    CONST robtarget Target_5570:=[[241.834905648,46.985576036,25.649683148],[0.692516726,0.060687774,-0.040025667,0.717729422],[-2,0,-1,0],[9E+09,9E+09,9E+09,9E+09,9E+09,9E+09]];
    CONST robtarget Target_5580:=[[234.328319461,46.702749675,25.84956623],[0.692516726,0.060687774,-0.040025667,0.717729422],[-2,0,-1,0],[9E+09,9E+09,9E+09,9E+09,9E+09,9E+09]];
    CONST robtarget Target_5590:=[[234.035172753,46.711233475,25.857420102],[0.692516726,0.060687774,-0.040025666,0.717729422],[-2,0,-1,0],[9E+09,9E+09,9E+09,9E+09,9E+09,9E+09]];
    CONST robtarget Target_5600:=[[233.779548655,46.760188453,25.864370937],[0.692516726,0.060687774,-0.040025666,0.717729422],[-2,0,-1,0],[9E+09,9E+09,9E+09,9E+09,9E+09,9E+09]];
    CONST robtarget Target_5610:=[[233.561447167,46.849614606,25.870418733],[0.692516726,0.060687774,-0.040025666,0.717729422],[-1,-1,0,0],[9E+09,9E+09,9E+09,9E+09,9E+09,9E+09]];
    CONST robtarget Target_5620:=[[233.380868291,46.979511937,25.875563491],[0.692516726,0.060687774,-0.040025667,0.717729422],[-1,-1,0,0],[9E+09,9E+09,9E+09,9E+09,9E+09,9E+09]];
    CONST robtarget Target_5630:=[[233.237812023,47.149880444,25.879805211],[0.692516726,0.060687774,-0.040025666,0.717729422],[-1,-1,0,0],[9E+09,9E+09,9E+09,9E+09,9E+09,9E+09]];
    CONST robtarget Target_5640:=[[233.132278367,47.360720127,25.883143893],[0.692516726,0.060687774,-0.040025666,0.717729422],[-1,-1,0,0],[9E+09,9E+09,9E+09,9E+09,9E+09,9E+09]];
    CONST robtarget Target_5650:=[[233.064267321,47.612030988,25.885579537],[0.692516726,0.060687774,-0.040025667,0.717729422],[-1,-1,0,0],[9E+09,9E+09,9E+09,9E+09,9E+09,9E+09]];
    CONST robtarget Target_5660:=[[233.033778885,47.903813024,25.887112143],[0.692516726,0.060687774,-0.040025667,0.717729422],[-1,-1,0,0],[9E+09,9E+09,9E+09,9E+09,9E+09,9E+09]];
    CONST robtarget Target_5670:=[[232.563911843,60.405319209,25.930427697],[0.692516726,0.060687774,-0.040025667,0.717729422],[-1,-1,0,0],[9E+09,9E+09,9E+09,9E+09,9E+09,9E+09]];
    CONST robtarget Target_5680:=[[232.572411908,60.698570219,25.930922129],[0.692516726,0.060687774,-0.040025667,0.717729422],[-1,-1,0,0],[9E+09,9E+09,9E+09,9E+09,9E+09,9E+09]];
    CONST robtarget Target_5690:=[[232.621366367,60.954288,25.930243251],[0.692516726,0.060687774,-0.040025666,0.717729422],[-1,-1,0,0],[9E+09,9E+09,9E+09,9E+09,9E+09,9E+09]];
    CONST robtarget Target_5700:=[[232.710775218,61.172472552,25.928391064],[0.692516726,0.060687774,-0.040025667,0.717729422],[-1,-1,0,0],[9E+09,9E+09,9E+09,9E+09,9E+09,9E+09]];
    CONST robtarget Target_5710:=[[232.840638463,61.353123873,25.925365567],[0.692516726,0.060687774,-0.040025666,0.717729422],[-1,-1,0,0],[9E+09,9E+09,9E+09,9E+09,9E+09,9E+09]];
    CONST robtarget Target_5720:=[[233.0109561,61.496241965,25.92116676],[0.692516726,0.060687774,-0.040025667,0.717729422],[-1,-1,0,0],[9E+09,9E+09,9E+09,9E+09,9E+09,9E+09]];
    CONST robtarget Target_5730:=[[233.221728132,61.601826826,25.915794643],[0.692516726,0.060687774,-0.040025667,0.717729422],[-1,-1,0,0],[9E+09,9E+09,9E+09,9E+09,9E+09,9E+09]];
    CONST robtarget Target_5740:=[[233.472954556,61.669878459,25.909249216],[0.692516726,0.060687774,-0.040025666,0.717729422],[-1,-1,0,0],[9E+09,9E+09,9E+09,9E+09,9E+09,9E+09]];
    CONST robtarget Target_5750:=[[233.764635372,61.700396861,25.90153048],[0.692516726,0.060687774,-0.040025667,0.717729422],[-2,0,-1,0],[9E+09,9E+09,9E+09,9E+09,9E+09,9E+09]];
    CONST robtarget Target_5760:=[[237.507531532,61.841418315,25.801865785],[0.692516726,0.060687774,-0.040025667,0.717729422],[-2,0,-1,0],[9E+09,9E+09,9E+09,9E+09,9E+09,9E+09]];
    CONST robtarget Target_5770:=[[237.80067824,61.832934515,25.794011913],[0.692516726,0.060687774,-0.040025666,0.717729422],[-2,0,-1,0],[9E+09,9E+09,9E+09,9E+09,9E+09,9E+09]];
    CONST robtarget Target_5780:=[[238.056302338,61.783979538,25.787061079],[0.692516726,0.060687774,-0.040025666,0.717729422],[-2,0,-1,0],[9E+09,9E+09,9E+09,9E+09,9E+09,9E+09]];
    CONST robtarget Target_5790:=[[238.274403825,61.694553384,25.781013283],[0.692516726,0.060687774,-0.040025666,0.717729422],[-2,0,-1,0],[9E+09,9E+09,9E+09,9E+09,9E+09,9E+09]];
    CONST robtarget Target_5800:=[[238.454982703,61.564656054,25.775868524],[0.692516726,0.060687774,-0.040025667,0.717729422],[-2,0,-1,0],[9E+09,9E+09,9E+09,9E+09,9E+09,9E+09]];
    CONST robtarget Target_5810:=[[238.598038969,61.394287547,25.771626804],[0.692516726,0.060687774,-0.040025666,0.717729422],[-2,0,-1,0],[9E+09,9E+09,9E+09,9E+09,9E+09,9E+09]];
    CONST robtarget Target_5820:=[[238.703572626,61.183447863,25.768288122],[0.692516726,0.060687774,-0.040025666,0.717729422],[-2,0,-1,0],[9E+09,9E+09,9E+09,9E+09,9E+09,9E+09]];
    CONST robtarget Target_5830:=[[238.771583672,60.932137002,25.765852478],[0.692516726,0.060687774,-0.040025667,0.717729422],[-2,0,-1,0],[9E+09,9E+09,9E+09,9E+09,9E+09,9E+09]];
    CONST robtarget Target_5840:=[[238.802072109,60.640354966,25.764319872],[0.692516726,0.060687774,-0.040025667,0.717729422],[-2,0,-1,0],[9E+09,9E+09,9E+09,9E+09,9E+09,9E+09]];
    CONST robtarget Target_5850:=[[238.793572042,60.347103955,25.76382544],[0.692516726,0.060687774,-0.040025667,0.717729422],[-2,0,-1,0],[9E+09,9E+09,9E+09,9E+09,9E+09,9E+09]];
    CONST robtarget Target_5860:=[[238.744617584,60.091386175,25.764504318],[0.692516726,0.060687774,-0.040025666,0.717729422],[-2,0,-1,0],[9E+09,9E+09,9E+09,9E+09,9E+09,9E+09]];
    CONST robtarget Target_5870:=[[238.655208732,59.873201624,25.766356505],[0.692516726,0.060687774,-0.040025667,0.717729422],[-2,0,-1,0],[9E+09,9E+09,9E+09,9E+09,9E+09,9E+09]];
    CONST robtarget Target_5880:=[[238.525345488,59.692550302,25.769382002],[0.692516726,0.060687774,-0.040025666,0.717729422],[-2,0,-1,0],[9E+09,9E+09,9E+09,9E+09,9E+09,9E+09]];
    CONST robtarget Target_5890:=[[238.35502785,59.549432211,25.773580809],[0.692516726,0.060687774,-0.040025667,0.717729422],[-2,0,-1,0],[9E+09,9E+09,9E+09,9E+09,9E+09,9E+09]];
    CONST robtarget Target_5900:=[[238.14425582,59.443847349,25.778952926],[0.692516726,0.060687774,-0.040025667,0.717729422],[-2,0,-1,0],[9E+09,9E+09,9E+09,9E+09,9E+09,9E+09]];
    CONST robtarget Target_5910:=[[237.893029395,59.375795717,25.785498353],[0.692516726,0.060687774,-0.040025666,0.717729422],[-2,0,-1,0],[9E+09,9E+09,9E+09,9E+09,9E+09,9E+09]];
    CONST robtarget Target_5920:=[[237.601348578,59.345277314,25.793217089],[0.692516726,0.060687774,-0.040025667,0.717729422],[-2,0,-1,0],[9E+09,9E+09,9E+09,9E+09,9E+09,9E+09]];
    CONST robtarget Target_5930:=[[236.800025002,59.419067101,-4.195988229],[0.692516726,0.060687774,-0.040025667,0.717729422],[-2,0,-1,0],[9E+09,9E+09,9E+09,9E+09,9E+09,9E+09]];
    CONST robtarget Target_5940:=[[225.383702429,63.988284743,-3.879696752],[0.692516726,0.060687774,-0.040025667,0.717729422],[0,0,0,0],[9E+09,9E+09,9E+09,9E+09,9E+09,9E+09]];
    CONST robtarget Target_5950:=[[226.185026006,63.914494956,26.109508566],[0.692516726,0.060687774,-0.040025667,0.717729422],[0,0,0,0],[9E+09,9E+09,9E+09,9E+09,9E+09,9E+09]];
    CONST robtarget Target_5960:=[[226.478172714,63.906011155,26.101654694],[0.692516726,0.060687774,-0.040025666,0.717729422],[0,0,0,0],[9E+09,9E+09,9E+09,9E+09,9E+09,9E+09]];
    CONST robtarget Target_5970:=[[226.733796812,63.857056178,26.094703859],[0.692516726,0.060687774,-0.040025666,0.717729422],[0,0,0,0],[9E+09,9E+09,9E+09,9E+09,9E+09,9E+09]];
    CONST robtarget Target_5980:=[[226.951898299,63.767630024,26.088656063],[0.692516726,0.060687774,-0.040025666,0.717729422],[0,0,0,0],[9E+09,9E+09,9E+09,9E+09,9E+09,9E+09]];
    CONST robtarget Target_5990:=[[227.132477177,63.637732694,26.083511305],[0.692516726,0.060687774,-0.040025667,0.717729422],[0,0,0,0],[9E+09,9E+09,9E+09,9E+09,9E+09,9E+09]];
    CONST robtarget Target_6000:=[[227.275533443,63.467364187,26.079269585],[0.692516726,0.060687774,-0.040025666,0.717729422],[0,0,0,0],[9E+09,9E+09,9E+09,9E+09,9E+09,9E+09]];
    CONST robtarget Target_6010:=[[227.3810671,63.256524503,26.075930903],[0.692516726,0.060687774,-0.040025666,0.717729422],[0,0,0,0],[9E+09,9E+09,9E+09,9E+09,9E+09,9E+09]];
    CONST robtarget Target_6020:=[[227.449078146,63.005213643,26.073495259],[0.692516726,0.060687774,-0.040025667,0.717729422],[0,0,0,0],[9E+09,9E+09,9E+09,9E+09,9E+09,9E+09]];
    CONST robtarget Target_6030:=[[227.479566583,62.713431606,26.071962653],[0.692516726,0.060687774,-0.040025667,0.717729422],[0,0,0,0],[9E+09,9E+09,9E+09,9E+09,9E+09,9E+09]];
    CONST robtarget Target_6040:=[[227.902525102,51.459995922,26.032971447],[0.692516726,0.060687774,-0.040025667,0.717729422],[0,0,0,0],[9E+09,9E+09,9E+09,9E+09,9E+09,9E+09]];
    CONST robtarget Target_6050:=[[227.899300134,50.944153551,26.031788366],[0.692516726,0.060687774,-0.040025666,0.717729422],[0,0,0,0],[9E+09,9E+09,9E+09,9E+09,9E+09,9E+09]];
    CONST robtarget Target_6060:=[[227.850143894,50.447085775,26.031878783],[0.692516726,0.060687774,-0.040025667,0.717729422],[0,0,0,0],[9E+09,9E+09,9E+09,9E+09,9E+09,9E+09]];
    CONST robtarget Target_6070:=[[227.755056379,49.968792596,26.033242698],[0.692516726,0.060687774,-0.040025666,0.717729422],[0,0,0,0],[9E+09,9E+09,9E+09,9E+09,9E+09,9E+09]];
    CONST robtarget Target_6080:=[[227.61403759,49.509274011,26.03588011],[0.692516726,0.060687774,-0.040025666,0.717729422],[0,0,0,0],[9E+09,9E+09,9E+09,9E+09,9E+09,9E+09]];
    CONST robtarget Target_6090:=[[227.427087528,49.068530022,26.03979102],[0.692516726,0.060687774,-0.040025666,0.717729422],[0,0,0,0],[9E+09,9E+09,9E+09,9E+09,9E+09,9E+09]];
    CONST robtarget Target_6100:=[[227.19420619,48.64656063,26.044975428],[0.692516726,0.060687774,-0.040025667,0.717729422],[0,0,0,0],[9E+09,9E+09,9E+09,9E+09,9E+09,9E+09]];
    CONST robtarget Target_6110:=[[226.915393579,48.243365833,26.051433334],[0.692516726,0.060687774,-0.040025666,0.717729422],[0,0,0,0],[9E+09,9E+09,9E+09,9E+09,9E+09,9E+09]];
    CONST robtarget Target_6120:=[[226.590649694,47.858945632,26.059164738],[0.692516726,0.060687774,-0.040025666,0.717729422],[0,0,0,0],[9E+09,9E+09,9E+09,9E+09,9E+09,9E+09]];
    CONST robtarget Target_6130:=[[226.231856695,47.506115899,26.067883677],[0.692516726,0.060687774,-0.040025666,0.717729422],[0,0,0,0],[9E+09,9E+09,9E+09,9E+09,9E+09,9E+09]];
    CONST robtarget Target_6140:=[[225.850896741,47.197692506,26.07730419],[0.692516726,0.060687774,-0.040025666,0.717729422],[0,0,0,0],[9E+09,9E+09,9E+09,9E+09,9E+09,9E+09]];
    CONST robtarget Target_6150:=[[225.447769833,46.933675455,26.087426276],[0.692516726,0.060687774,-0.040025667,0.717729422],[0,0,0,0],[9E+09,9E+09,9E+09,9E+09,9E+09,9E+09]];
    CONST robtarget Target_6160:=[[225.022475972,46.714064745,26.098249937],[0.692516726,0.060687774,-0.040025667,0.717729422],[0,0,0,0],[9E+09,9E+09,9E+09,9E+09,9E+09,9E+09]];
    CONST robtarget Target_6170:=[[224.575015155,46.538860376,26.109775171],[0.692516726,0.060687774,-0.040025667,0.717729422],[0,0,0,0],[9E+09,9E+09,9E+09,9E+09,9E+09,9E+09]];
    CONST robtarget Target_6180:=[[224.105387385,46.408062347,26.122001978],[0.692516726,0.060687774,-0.040025667,0.717729422],[0,0,0,0],[9E+09,9E+09,9E+09,9E+09,9E+09,9E+09]];
    CONST robtarget Target_6190:=[[223.61359266,46.321670659,26.13493036],[0.692516726,0.060687774,-0.040025667,0.717729422],[0,0,0,0],[9E+09,9E+09,9E+09,9E+09,9E+09,9E+09]];
    CONST robtarget Target_6200:=[[223.099630982,46.279685313,26.148560315],[0.692516726,0.060687774,-0.040025667,0.717729422],[0,0,0,0],[9E+09,9E+09,9E+09,9E+09,9E+09,9E+09]];
    CONST robtarget Target_6210:=[[216.840676848,46.043866104,26.315221832],[0.692516726,0.060687774,-0.040025667,0.717729422],[0,0,0,0],[9E+09,9E+09,9E+09,9E+09,9E+09,9E+09]];
    CONST robtarget Target_6220:=[[216.547530141,46.052349904,26.323075704],[0.692516726,0.060687774,-0.040025666,0.717729422],[0,0,0,0],[9E+09,9E+09,9E+09,9E+09,9E+09,9E+09]];
    CONST robtarget Target_6230:=[[216.291906042,46.101304881,26.330026538],[0.692516726,0.060687774,-0.040025666,0.717729422],[0,0,0,0],[9E+09,9E+09,9E+09,9E+09,9E+09,9E+09]];
    CONST robtarget Target_6240:=[[216.073804554,46.190731035,26.336074335],[0.692516726,0.060687774,-0.040025666,0.717729422],[0,0,0,0],[9E+09,9E+09,9E+09,9E+09,9E+09,9E+09]];
    CONST robtarget Target_6250:=[[215.893225678,46.320628365,26.341219093],[0.692516726,0.060687774,-0.040025667,0.717729422],[0,0,0,0],[9E+09,9E+09,9E+09,9E+09,9E+09,9E+09]];
    CONST robtarget Target_6260:=[[215.75016941,46.490996873,26.345460813],[0.692516726,0.060687774,-0.040025666,0.717729422],[0,0,0,0],[9E+09,9E+09,9E+09,9E+09,9E+09,9E+09]];
    CONST robtarget Target_6270:=[[215.644635754,46.701836556,26.348799495],[0.692516726,0.060687774,-0.040025666,0.717729422],[0,0,0,0],[9E+09,9E+09,9E+09,9E+09,9E+09,9E+09]];
    CONST robtarget Target_6280:=[[215.576624708,46.953147417,26.351235139],[0.692516726,0.060687774,-0.040025667,0.717729422],[0,0,0,0],[9E+09,9E+09,9E+09,9E+09,9E+09,9E+09]];
    CONST robtarget Target_6290:=[[215.546136272,47.244929453,26.352767745],[0.692516726,0.060687774,-0.040025667,0.717729422],[0,0,0,0],[9E+09,9E+09,9E+09,9E+09,9E+09,9E+09]];
    CONST robtarget Target_6300:=[[214.982452183,62.24257664,26.404731995],[0.692516726,0.060687774,-0.040025667,0.717729422],[0,0,0,0],[9E+09,9E+09,9E+09,9E+09,9E+09,9E+09]];
    CONST robtarget Target_6310:=[[214.990952248,62.53582765,26.405226427],[0.692516726,0.060687774,-0.040025667,0.717729422],[0,0,0,0],[9E+09,9E+09,9E+09,9E+09,9E+09,9E+09]];
    CONST robtarget Target_6320:=[[215.039906707,62.791545431,26.404547549],[0.692516726,0.060687774,-0.040025666,0.717729422],[0,0,0,0],[9E+09,9E+09,9E+09,9E+09,9E+09,9E+09]];
    CONST robtarget Target_6330:=[[215.129315559,63.009729982,26.402695362],[0.692516726,0.060687774,-0.040025667,0.717729422],[0,0,0,0],[9E+09,9E+09,9E+09,9E+09,9E+09,9E+09]];
    CONST robtarget Target_6340:=[[215.259178804,63.190381304,26.399669865],[0.692516726,0.060687774,-0.040025666,0.717729422],[0,0,0,0],[9E+09,9E+09,9E+09,9E+09,9E+09,9E+09]];
    CONST robtarget Target_6350:=[[215.429496441,63.333499395,26.395471058],[0.692516726,0.060687774,-0.040025667,0.717729422],[0,0,0,0],[9E+09,9E+09,9E+09,9E+09,9E+09,9E+09]];
    CONST robtarget Target_6360:=[[215.640268472,63.439084257,26.390098941],[0.692516726,0.060687774,-0.040025667,0.717729422],[0,0,0,0],[9E+09,9E+09,9E+09,9E+09,9E+09,9E+09]];
    CONST robtarget Target_6370:=[[215.891494896,63.507135889,26.383553514],[0.692516726,0.060687774,-0.040025666,0.717729422],[0,0,0,0],[9E+09,9E+09,9E+09,9E+09,9E+09,9E+09]];
    CONST robtarget Target_6380:=[[216.183175712,63.537654292,26.375834778],[0.692516726,0.060687774,-0.040025667,0.717729422],[0,0,0,0],[9E+09,9E+09,9E+09,9E+09,9E+09,9E+09]];
    CONST robtarget Target_6390:=[[215.381852135,63.61144408,-3.61337054],[0.692516726,0.060687774,-0.040025667,0.717729422],[0,0,0,0],[9E+09,9E+09,9E+09,9E+09,9E+09,9E+09]];
    CONST robtarget Target_6400:=[[197.988026569,60.456419506,-3.156363634],[0.692516726,0.060687774,-0.040025667,0.717729422],[0,0,0,0],[9E+09,9E+09,9E+09,9E+09,9E+09,9E+09]];
    CONST robtarget Target_6410:=[[198.789350146,60.382629718,26.832841684],[0.692516726,0.060687774,-0.040025667,0.717729422],[0,0,0,0],[9E+09,9E+09,9E+09,9E+09,9E+09,9E+09]];
    CONST robtarget Target_6420:=[[198.793455963,60.5504059,26.833144795],[0.692516726,0.060687774,-0.040025667,0.717729422],[0,0,0,0],[9E+09,9E+09,9E+09,9E+09,9E+09,9E+09]];
    CONST robtarget Target_6430:=[[198.818673257,60.710515057,26.832864935],[0.692516726,0.060687774,-0.040025667,0.717729422],[0,0,0,0],[9E+09,9E+09,9E+09,9E+09,9E+09,9E+09]];
    CONST robtarget Target_6440:=[[198.865002028,60.862957189,26.832002102],[0.692516726,0.060687774,-0.040025667,0.717729422],[0,0,0,0],[9E+09,9E+09,9E+09,9E+09,9E+09,9E+09]];
    CONST robtarget Target_6450:=[[198.932442278,61.007732296,26.830556297],[0.692516726,0.060687774,-0.040025666,0.717729422],[0,0,0,0],[9E+09,9E+09,9E+09,9E+09,9E+09,9E+09]];
    CONST robtarget Target_6460:=[[199.020994004,61.144840378,26.82852752],[0.692516726,0.060687774,-0.040025666,0.717729422],[0,0,0,0],[9E+09,9E+09,9E+09,9E+09,9E+09,9E+09]];
    CONST robtarget Target_6470:=[[199.130657206,61.274281435,26.825915771],[0.692516726,0.060687774,-0.040025667,0.717729422],[0,0,0,0],[9E+09,9E+09,9E+09,9E+09,9E+09,9E+09]];
    CONST robtarget Target_6480:=[[199.261431888,61.396055468,26.82272105],[0.692516726,0.060687774,-0.040025666,0.717729422],[0,0,0,0],[9E+09,9E+09,9E+09,9E+09,9E+09,9E+09]];
    CONST robtarget Target_6490:=[[199.413318046,61.510162475,26.818943356],[0.692516726,0.060687774,-0.040025666,0.717729422],[0,0,0,0],[9E+09,9E+09,9E+09,9E+09,9E+09,9E+09]];
    CONST robtarget Target_6500:=[[199.961359249,61.853034903,26.805143129],[0.692516726,0.060687774,-0.040025666,0.717729422],[0,0,0,0],[9E+09,9E+09,9E+09,9E+09,9E+09,9E+09]];
    CONST robtarget Target_6510:=[[200.529207568,62.15369043,26.790709771],[0.692516726,0.060687774,-0.040025667,0.717729422],[0,0,0,0],[9E+09,9E+09,9E+09,9E+09,9E+09,9E+09]];
    CONST robtarget Target_6520:=[[201.116863,62.412129053,26.775643282],[0.692516726,0.060687774,-0.040025667,0.717729422],[0,0,0,0],[9E+09,9E+09,9E+09,9E+09,9E+09,9E+09]];
    CONST robtarget Target_6530:=[[201.724325548,62.628350774,26.759943663],[0.692516726,0.060687774,-0.040025667,0.717729422],[0,0,0,0],[9E+09,9E+09,9E+09,9E+09,9E+09,9E+09]];
    CONST robtarget Target_6540:=[[202.351595209,62.802355592,26.743610913],[0.692516726,0.060687774,-0.040025667,0.717729422],[0,0,0,0],[9E+09,9E+09,9E+09,9E+09,9E+09,9E+09]];
    CONST robtarget Target_6550:=[[202.998671986,62.934143508,26.726645033],[0.692516726,0.060687774,-0.040025666,0.717729422],[0,0,0,0],[9E+09,9E+09,9E+09,9E+09,9E+09,9E+09]];
    CONST robtarget Target_6560:=[[203.665555877,63.023714521,26.709046021],[0.692516726,0.060687774,-0.040025666,0.717729422],[0,0,0,0],[9E+09,9E+09,9E+09,9E+09,9E+09,9E+09]];
    CONST robtarget Target_6570:=[[204.352246883,63.071068632,26.69081388],[0.692516726,0.060687774,-0.040025667,0.717729422],[0,0,0,0],[9E+09,9E+09,9E+09,9E+09,9E+09,9E+09]];
    CONST robtarget Target_6580:=[[204.912655358,63.076234743,26.675852252],[0.692516726,0.060687774,-0.040025667,0.717729422],[0,0,0,0],[9E+09,9E+09,9E+09,9E+09,9E+09,9E+09]];
    CONST robtarget Target_6590:=[[205.450218069,63.048643188,26.661420471],[0.692516726,0.060687774,-0.040025667,0.717729422],[0,0,0,0],[9E+09,9E+09,9E+09,9E+09,9E+09,9E+09]];
    CONST robtarget Target_6600:=[[205.964935015,62.988293967,26.647518536],[0.692516726,0.060687774,-0.040025667,0.717729422],[0,0,0,0],[9E+09,9E+09,9E+09,9E+09,9E+09,9E+09]];
    CONST robtarget Target_6610:=[[206.456806196,62.895187079,26.634146447],[0.692516726,0.060687774,-0.040025667,0.717729422],[0,0,0,0],[9E+09,9E+09,9E+09,9E+09,9E+09,9E+09]];
    CONST robtarget Target_6620:=[[206.925831612,62.769322526,26.621304205],[0.692516726,0.060687774,-0.040025666,0.717729422],[0,0,0,0],[9E+09,9E+09,9E+09,9E+09,9E+09,9E+09]];
    CONST robtarget Target_6630:=[[207.372011264,62.610700306,26.608991809],[0.692516726,0.060687774,-0.040025667,0.717729422],[0,0,0,0],[9E+09,9E+09,9E+09,9E+09,9E+09,9E+09]];
    CONST robtarget Target_6640:=[[207.795345151,62.41932042,26.597209259],[0.692516726,0.060687774,-0.040025666,0.717729422],[0,0,0,0],[9E+09,9E+09,9E+09,9E+09,9E+09,9E+09]];
    CONST robtarget Target_6650:=[[208.195833273,62.195182868,26.585956556],[0.692516726,0.060687774,-0.040025667,0.717729422],[0,0,0,0],[9E+09,9E+09,9E+09,9E+09,9E+09,9E+09]];
    CONST robtarget Target_6660:=[[208.626662365,61.899606744,26.573717351],[0.692516726,0.060687774,-0.040025667,0.717729422],[0,0,0,0],[9E+09,9E+09,9E+09,9E+09,9E+09,9E+09]];
    CONST robtarget Target_6670:=[[209.002731788,61.572023403,26.562862592],[0.692516726,0.060687774,-0.040025666,0.717729422],[0,0,0,0],[9E+09,9E+09,9E+09,9E+09,9E+09,9E+09]];
    CONST robtarget Target_6680:=[[209.324041543,61.212432844,26.553392278],[0.692516726,0.060687774,-0.040025667,0.717729422],[0,0,0,0],[9E+09,9E+09,9E+09,9E+09,9E+09,9E+09]];
    CONST robtarget Target_6690:=[[209.590591627,60.820835066,26.545306409],[0.692516726,0.060687774,-0.040025667,0.717729422],[0,0,0,0],[9E+09,9E+09,9E+09,9E+09,9E+09,9E+09]];
    CONST robtarget Target_6700:=[[209.802382044,60.397230073,26.538604985],[0.692516726,0.060687774,-0.040025667,0.717729422],[0,0,0,0],[9E+09,9E+09,9E+09,9E+09,9E+09,9E+09]];
    CONST robtarget Target_6710:=[[209.959412791,59.94161786,26.533288007],[0.692516726,0.060687774,-0.040025667,0.717729422],[0,0,0,0],[9E+09,9E+09,9E+09,9E+09,9E+09,9E+09]];
    CONST robtarget Target_6720:=[[210.061683869,59.45399843,26.529355473],[0.692516726,0.060687774,-0.040025667,0.717729422],[0,0,0,0],[9E+09,9E+09,9E+09,9E+09,9E+09,9E+09]];
    CONST robtarget Target_6730:=[[210.109195278,58.934371782,26.526807384],[0.692516726,0.060687774,-0.040025667,0.717729422],[0,0,0,0],[9E+09,9E+09,9E+09,9E+09,9E+09,9E+09]];
    CONST robtarget Target_6740:=[[210.112043833,58.596713676,26.525900447],[0.692516726,0.060687774,-0.040025667,0.717729422],[0,0,0,0],[9E+09,9E+09,9E+09,9E+09,9E+09,9E+09]];
    CONST robtarget Target_6750:=[[210.094789809,58.270178132,26.525558026],[0.692516726,0.060687774,-0.040025667,0.717729422],[0,0,0,0],[9E+09,9E+09,9E+09,9E+09,9E+09,9E+09]];
    CONST robtarget Target_6760:=[[210.057433208,57.954765151,26.525780121],[0.692516726,0.060687774,-0.040025667,0.717729422],[0,0,0,0],[9E+09,9E+09,9E+09,9E+09,9E+09,9E+09]];
    CONST robtarget Target_6770:=[[209.999974028,57.650474732,26.526566733],[0.692516726,0.060687774,-0.040025667,0.717729422],[0,0,0,0],[9E+09,9E+09,9E+09,9E+09,9E+09,9E+09]];
    CONST robtarget Target_6780:=[[209.92241227,57.357306876,26.527917862],[0.692516726,0.060687774,-0.040025667,0.717729422],[0,0,0,0],[9E+09,9E+09,9E+09,9E+09,9E+09,9E+09]];
    CONST robtarget Target_6790:=[[209.824747934,57.075261584,26.529833507],[0.692516726,0.060687774,-0.040025666,0.717729422],[0,0,0,0],[9E+09,9E+09,9E+09,9E+09,9E+09,9E+09]];
    CONST robtarget Target_6800:=[[209.706981019,56.804338853,26.532313669],[0.692516726,0.060687774,-0.040025667,0.717729422],[0,0,0,0],[9E+09,9E+09,9E+09,9E+09,9E+09,9E+09]];
    CONST robtarget Target_6810:=[[209.569111527,56.544538685,26.535358347],[0.692516726,0.060687774,-0.040025667,0.717729422],[0,0,0,0],[9E+09,9E+09,9E+09,9E+09,9E+09,9E+09]];
    CONST robtarget Target_6820:=[[209.411139456,56.29586108,26.538967541],[0.692516726,0.060687774,-0.040025666,0.717729422],[0,0,0,0],[9E+09,9E+09,9E+09,9E+09,9E+09,9E+09]];
    CONST robtarget Target_6830:=[[209.233064807,56.058306038,26.543141252],[0.692516726,0.060687774,-0.040025666,0.717729422],[0,0,0,0],[9E+09,9E+09,9E+09,9E+09,9E+09,9E+09]];
    CONST robtarget Target_6840:=[[209.034887579,55.831873558,26.54787948],[0.692516726,0.060687774,-0.040025667,0.717729422],[0,0,0,0],[9E+09,9E+09,9E+09,9E+09,9E+09,9E+09]];
    CONST robtarget Target_6850:=[[208.816607774,55.61656364,26.553182224],[0.692516726,0.060687774,-0.040025666,0.717729422],[0,0,0,0],[9E+09,9E+09,9E+09,9E+09,9E+09,9E+09]];
    CONST robtarget Target_6860:=[[208.578225391,55.412376287,26.559049485],[0.692516726,0.060687774,-0.040025667,0.717729422],[0,0,0,0],[9E+09,9E+09,9E+09,9E+09,9E+09,9E+09]];
    CONST robtarget Target_6870:=[[208.319740428,55.219311494,26.565481262],[0.692516726,0.060687774,-0.040025667,0.717729422],[0,0,0,0],[9E+09,9E+09,9E+09,9E+09,9E+09,9E+09]];
    CONST robtarget Target_6880:=[[208.041152888,55.037369265,26.572477555],[0.692516726,0.060687774,-0.040025666,0.717729422],[0,0,0,0],[9E+09,9E+09,9E+09,9E+09,9E+09,9E+09]];
    CONST robtarget Target_6890:=[[207.74246277,54.866549599,26.580038365],[0.692516726,0.060687774,-0.040025666,0.717729422],[0,0,0,0],[9E+09,9E+09,9E+09,9E+09,9E+09,9E+09]];
    CONST robtarget Target_6900:=[[201.432865387,51.545888867,26.740462699],[0.692516726,0.060687774,-0.040025667,0.717729422],[0,0,0,0],[9E+09,9E+09,9E+09,9E+09,9E+09,9E+09]];
    CONST robtarget Target_6910:=[[201.189590898,51.39611623,26.746594569],[0.692516726,0.060687774,-0.040025667,0.717729422],[0,0,0,0],[9E+09,9E+09,9E+09,9E+09,9E+09,9E+09]];
    CONST robtarget Target_6920:=[[200.980238444,51.226791045,26.751771918],[0.692516726,0.060687774,-0.040025667,0.717729422],[0,0,0,0],[9E+09,9E+09,9E+09,9E+09,9E+09,9E+09]];
    CONST robtarget Target_6930:=[[200.804808025,51.037913312,26.755994747],[0.692516726,0.060687774,-0.040025667,0.717729422],[0,0,0,0],[9E+09,9E+09,9E+09,9E+09,9E+09,9E+09]];
    CONST robtarget Target_6940:=[[200.663299641,50.829483032,26.759263056],[0.692516726,0.060687774,-0.040025667,0.717729422],[0,0,0,0],[9E+09,9E+09,9E+09,9E+09,9E+09,9E+09]];
    CONST robtarget Target_6950:=[[200.555713292,50.601500205,26.761576844],[0.692516726,0.060687774,-0.040025666,0.717729422],[0,0,0,0],[9E+09,9E+09,9E+09,9E+09,9E+09,9E+09]];
    CONST robtarget Target_6960:=[[200.482048978,50.35396483,26.762936112],[0.692516726,0.060687774,-0.040025667,0.717729422],[0,0,0,0],[9E+09,9E+09,9E+09,9E+09,9E+09,9E+09]];
    CONST robtarget Target_6970:=[[200.4423067,50.086876907,26.76334086],[0.692516726,0.060687774,-0.040025667,0.717729422],[0,0,0,0],[9E+09,9E+09,9E+09,9E+09,9E+09,9E+09]];
    CONST robtarget Target_6980:=[[200.436486457,49.800236437,26.762791087],[0.692516726,0.060687774,-0.040025667,0.717729422],[0,0,0,0],[9E+09,9E+09,9E+09,9E+09,9E+09,9E+09]];
    CONST robtarget Target_6990:=[[200.457434535,49.574004366,26.761674692],[0.692516726,0.060687774,-0.040025667,0.717729422],[0,0,0,0],[9E+09,9E+09,9E+09,9E+09,9E+09,9E+09]];
    CONST robtarget Target_7000:=[[200.502688074,49.363334593,26.759947137],[0.692516726,0.060687774,-0.040025667,0.717729422],[0,0,0,0],[9E+09,9E+09,9E+09,9E+09,9E+09,9E+09]];
    CONST robtarget Target_7010:=[[200.572247074,49.168227116,26.757608422],[0.692516726,0.060687774,-0.040025666,0.717729422],[0,0,0,0],[9E+09,9E+09,9E+09,9E+09,9E+09,9E+09]];
    CONST robtarget Target_7020:=[[200.666111534,48.988681936,26.754658547],[0.692516726,0.060687774,-0.040025666,0.717729422],[0,0,0,0],[9E+09,9E+09,9E+09,9E+09,9E+09,9E+09]];
    CONST robtarget Target_7030:=[[200.784281454,48.824699052,26.751097512],[0.692516726,0.060687774,-0.040025666,0.717729422],[0,0,0,0],[9E+09,9E+09,9E+09,9E+09,9E+09,9E+09]];
    CONST robtarget Target_7040:=[[200.926756835,48.676278466,26.746925317],[0.692516726,0.060687774,-0.040025667,0.717729422],[0,0,0,0],[9E+09,9E+09,9E+09,9E+09,9E+09,9E+09]];
    CONST robtarget Target_7050:=[[201.093537677,48.543420176,26.742141963],[0.692516726,0.060687774,-0.040025667,0.717729422],[0,0,0,0],[9E+09,9E+09,9E+09,9E+09,9E+09,9E+09]];
    CONST robtarget Target_7060:=[[201.284623979,48.426124182,26.736747448],[0.692516726,0.060687774,-0.040025667,0.717729422],[0,0,0,0],[9E+09,9E+09,9E+09,9E+09,9E+09,9E+09]];
    CONST robtarget Target_7070:=[[201.500015743,48.324390486,26.730741774],[0.692516726,0.060687774,-0.040025666,0.717729422],[0,0,0,0],[9E+09,9E+09,9E+09,9E+09,9E+09,9E+09]];
    CONST robtarget Target_7080:=[[201.739712966,48.238219087,26.724124939],[0.692516726,0.060687774,-0.040025667,0.717729422],[0,0,0,0],[9E+09,9E+09,9E+09,9E+09,9E+09,9E+09]];
    CONST robtarget Target_7090:=[[202.00371565,48.167609984,26.716896945],[0.692516726,0.060687774,-0.040025666,0.717729422],[0,0,0,0],[9E+09,9E+09,9E+09,9E+09,9E+09,9E+09]];
    CONST robtarget Target_7100:=[[202.292023794,48.112563178,26.709057791],[0.692516726,0.060687774,-0.040025666,0.717729422],[0,0,0,0],[9E+09,9E+09,9E+09,9E+09,9E+09,9E+09]];
    CONST robtarget Target_7110:=[[202.604637399,48.073078669,26.700607476],[0.692516726,0.060687774,-0.040025667,0.717729422],[0,0,0,0],[9E+09,9E+09,9E+09,9E+09,9E+09,9E+09]];
    CONST robtarget Target_7120:=[[202.941556464,48.049156456,26.691546002],[0.692516726,0.060687774,-0.040025666,0.717729422],[0,0,0,0],[9E+09,9E+09,9E+09,9E+09,9E+09,9E+09]];
    CONST robtarget Target_7130:=[[203.302780991,48.04079654,26.681873368],[0.692516726,0.060687774,-0.040025666,0.717729422],[0,0,0,0],[9E+09,9E+09,9E+09,9E+09,9E+09,9E+09]];
    CONST robtarget Target_7140:=[[203.688310978,48.047998921,26.671589575],[0.692516726,0.060687774,-0.040025667,0.717729422],[0,0,0,0],[9E+09,9E+09,9E+09,9E+09,9E+09,9E+09]];
    CONST robtarget Target_7150:=[[204.503395292,48.107351049,26.649956234],[0.692516726,0.060687774,-0.040025666,0.717729422],[0,0,0,0],[9E+09,9E+09,9E+09,9E+09,9E+09,9E+09]];
    CONST robtarget Target_7160:=[[205.326726566,48.224298133,26.628244246],[0.692516726,0.060687774,-0.040025667,0.717729422],[0,0,0,0],[9E+09,9E+09,9E+09,9E+09,9E+09,9E+09]];
    CONST robtarget Target_7170:=[[206.158304801,48.398840175,26.606453611],[0.692516726,0.060687774,-0.040025666,0.717729422],[0,0,0,0],[9E+09,9E+09,9E+09,9E+09,9E+09,9E+09]];
    CONST robtarget Target_7180:=[[206.998129994,48.630977175,26.584584329],[0.692516726,0.060687774,-0.040025667,0.717729422],[0,0,0,0],[9E+09,9E+09,9E+09,9E+09,9E+09,9E+09]];
    CONST robtarget Target_7190:=[[207.537450548,48.85960352,26.570736013],[0.692516726,0.060687774,-0.040025667,0.717729422],[0,0,0,0],[9E+09,9E+09,9E+09,9E+09,9E+09,9E+09]];
    CONST robtarget Target_7200:=[[208.007373606,49.064784538,26.558684338],[0.692516726,0.060687774,-0.040025666,0.717729422],[0,0,0,0],[9E+09,9E+09,9E+09,9E+09,9E+09,9E+09]];
    CONST robtarget Target_7210:=[[208.40789917,49.246520227,26.548429303],[0.692516726,0.060687774,-0.040025667,0.717729422],[0,0,0,0],[9E+09,9E+09,9E+09,9E+09,9E+09,9E+09]];
    CONST robtarget Target_7220:=[[208.73902724,49.40481059,26.539970909],[0.692516726,0.060687774,-0.040025666,0.717729422],[0,0,0,0],[9E+09,9E+09,9E+09,9E+09,9E+09,9E+09]];
    CONST robtarget Target_7230:=[[208.970612824,49.476027956,26.533958083],[0.692516726,0.060687774,-0.040025666,0.717729422],[0,0,0,0],[9E+09,9E+09,9E+09,9E+09,9E+09,9E+09]];
    CONST robtarget Target_7240:=[[209.214158959,49.506034699,26.527524266],[0.692516726,0.060687774,-0.040025667,0.717729422],[0,0,0,0],[9E+09,9E+09,9E+09,9E+09,9E+09,9E+09]];
    CONST robtarget Target_7250:=[[209.456742772,49.492391048,26.521008758],[0.692516726,0.060687774,-0.040025666,0.717729422],[0,0,0,0],[9E+09,9E+09,9E+09,9E+09,9E+09,9E+09]];
    CONST robtarget Target_7260:=[[209.685441392,49.432657239,26.514750862],[0.692516726,0.060687774,-0.040025666,0.717729422],[0,0,0,0],[9E+09,9E+09,9E+09,9E+09,9E+09,9E+09]];
    CONST robtarget Target_7270:=[[209.900254818,49.326833271,26.508750577],[0.692516726,0.060687774,-0.040025666,0.717729422],[0,0,0,0],[9E+09,9E+09,9E+09,9E+09,9E+09,9E+09]];
    CONST robtarget Target_7280:=[[210.101183049,49.174919142,26.503007902],[0.692516726,0.060687774,-0.040025666,0.717729422],[0,0,0,0],[9E+09,9E+09,9E+09,9E+09,9E+09,9E+09]];
    CONST robtarget Target_7290:=[[210.272142055,48.989327998,26.497983154],[0.692516726,0.060687774,-0.040025666,0.717729422],[0,0,0,0],[9E+09,9E+09,9E+09,9E+09,9E+09,9E+09]];
    CONST robtarget Target_7300:=[[210.397047805,48.782472985,26.494136646],[0.692516726,0.060687774,-0.040025667,0.717729422],[0,0,0,0],[9E+09,9E+09,9E+09,9E+09,9E+09,9E+09]];
    CONST robtarget Target_7310:=[[210.475900298,48.554354102,26.491468379],[0.692516726,0.060687774,-0.040025667,0.717729422],[0,0,0,0],[9E+09,9E+09,9E+09,9E+09,9E+09,9E+09]];
    CONST robtarget Target_7320:=[[210.508699535,48.304971349,26.489978353],[0.692516726,0.060687774,-0.040025667,0.717729422],[0,0,0,0],[9E+09,9E+09,9E+09,9E+09,9E+09,9E+09]];
    CONST robtarget Target_7330:=[[209.707375959,48.378761136,-3.499226965],[0.692516726,0.060687774,-0.040025667,0.717729422],[0,0,0,0],[9E+09,9E+09,9E+09,9E+09,9E+09,9E+09]];
    CONST robtarget Target_7340:=[[187.631701957,70.064926304,-2.85599633],[0.692516726,0.060687774,-0.040025667,0.717729422],[0,0,0,0],[9E+09,9E+09,9E+09,9E+09,9E+09,9E+09]];
    CONST robtarget Target_7350:=[[188.433025534,69.991136516,27.133208988],[0.692516726,0.060687774,-0.040025667,0.717729422],[0,0,0,0],[9E+09,9E+09,9E+09,9E+09,9E+09,9E+09]];
    CONST robtarget Target_7360:=[[188.726172242,69.982652715,27.125355116],[0.692516726,0.060687774,-0.040025666,0.717729422],[0,0,0,0],[9E+09,9E+09,9E+09,9E+09,9E+09,9E+09]];
    CONST robtarget Target_7370:=[[188.981796339,69.933697738,27.118404281],[0.692516726,0.060687774,-0.040025666,0.717729422],[0,0,0,0],[9E+09,9E+09,9E+09,9E+09,9E+09,9E+09]];
    CONST robtarget Target_7380:=[[189.199897827,69.844271584,27.112356485],[0.692516726,0.060687774,-0.040025666,0.717729422],[0,0,0,0],[9E+09,9E+09,9E+09,9E+09,9E+09,9E+09]];
    CONST robtarget Target_7390:=[[189.380476704,69.714374254,27.107211727],[0.692516726,0.060687774,-0.040025667,0.717729422],[0,0,0,0],[9E+09,9E+09,9E+09,9E+09,9E+09,9E+09]];
    CONST robtarget Target_7400:=[[189.523532971,69.544005747,27.102970007],[0.692516726,0.060687774,-0.040025666,0.717729422],[0,0,0,0],[9E+09,9E+09,9E+09,9E+09,9E+09,9E+09]];
    CONST robtarget Target_7410:=[[189.629066628,69.333166063,27.099631325],[0.692516726,0.060687774,-0.040025666,0.717729422],[0,0,0,0],[9E+09,9E+09,9E+09,9E+09,9E+09,9E+09]];
    CONST robtarget Target_7420:=[[189.697077674,69.081855203,27.097195681],[0.692516726,0.060687774,-0.040025667,0.717729422],[0,0,0,0],[9E+09,9E+09,9E+09,9E+09,9E+09,9E+09]];
    CONST robtarget Target_7430:=[[189.727566111,68.790073166,27.095663075],[0.692516726,0.060687774,-0.040025667,0.717729422],[0,0,0,0],[9E+09,9E+09,9E+09,9E+09,9E+09,9E+09]];
    CONST robtarget Target_7440:=[[189.962108727,62.549720662,27.074041334],[0.692516726,0.060687774,-0.040025667,0.717729422],[0,0,0,0],[9E+09,9E+09,9E+09,9E+09,9E+09,9E+09]];
    CONST robtarget Target_7450:=[[191.20974078,62.596727813,27.040819769],[0.692516726,0.060687774,-0.040025667,0.717729422],[0,0,0,0],[9E+09,9E+09,9E+09,9E+09,9E+09,9E+09]];
    CONST robtarget Target_7460:=[[191.502887488,62.588244012,27.032965897],[0.692516726,0.060687774,-0.040025666,0.717729422],[0,0,0,0],[9E+09,9E+09,9E+09,9E+09,9E+09,9E+09]];
    CONST robtarget Target_7470:=[[191.758511587,62.539289035,27.026015063],[0.692516726,0.060687774,-0.040025666,0.717729422],[0,0,0,0],[9E+09,9E+09,9E+09,9E+09,9E+09,9E+09]];
    CONST robtarget Target_7480:=[[191.976613074,62.449862881,27.019967267],[0.692516726,0.060687774,-0.040025666,0.717729422],[0,0,0,0],[9E+09,9E+09,9E+09,9E+09,9E+09,9E+09]];
    CONST robtarget Target_7490:=[[192.157191951,62.319965551,27.014822509],[0.692516726,0.060687774,-0.040025667,0.717729422],[0,0,0,0],[9E+09,9E+09,9E+09,9E+09,9E+09,9E+09]];
    CONST robtarget Target_7500:=[[192.300248218,62.149597044,27.010580789],[0.692516726,0.060687774,-0.040025666,0.717729422],[0,0,0,0],[9E+09,9E+09,9E+09,9E+09,9E+09,9E+09]];
    CONST robtarget Target_7510:=[[192.405781875,61.93875736,27.007242106],[0.692516726,0.060687774,-0.040025666,0.717729422],[0,0,0,0],[9E+09,9E+09,9E+09,9E+09,9E+09,9E+09]];
    CONST robtarget Target_7520:=[[192.47379292,61.6874465,27.004806462],[0.692516726,0.060687774,-0.040025667,0.717729422],[0,0,0,0],[9E+09,9E+09,9E+09,9E+09,9E+09,9E+09]];
    CONST robtarget Target_7530:=[[192.504281357,61.395664463,27.003273856],[0.692516726,0.060687774,-0.040025667,0.717729422],[0,0,0,0],[9E+09,9E+09,9E+09,9E+09,9E+09,9E+09]];
    CONST robtarget Target_7540:=[[192.495781291,61.102413452,27.002779424],[0.692516726,0.060687774,-0.040025667,0.717729422],[0,0,0,0],[9E+09,9E+09,9E+09,9E+09,9E+09,9E+09]];
    CONST robtarget Target_7550:=[[192.446826833,60.846695672,27.003458302],[0.692516726,0.060687774,-0.040025666,0.717729422],[0,0,0,0],[9E+09,9E+09,9E+09,9E+09,9E+09,9E+09]];
    CONST robtarget Target_7560:=[[192.35741798,60.628511121,27.005310489],[0.692516726,0.060687774,-0.040025667,0.717729422],[0,0,0,0],[9E+09,9E+09,9E+09,9E+09,9E+09,9E+09]];
    CONST robtarget Target_7570:=[[192.227554736,60.4478598,27.008335986],[0.692516726,0.060687774,-0.040025666,0.717729422],[0,0,0,0],[9E+09,9E+09,9E+09,9E+09,9E+09,9E+09]];
    CONST robtarget Target_7580:=[[192.057237098,60.304741708,27.012534793],[0.692516726,0.060687774,-0.040025667,0.717729422],[0,0,0,0],[9E+09,9E+09,9E+09,9E+09,9E+09,9E+09]];
    CONST robtarget Target_7590:=[[191.846465068,60.199156846,27.01790691],[0.692516726,0.060687774,-0.040025667,0.717729422],[0,0,0,0],[9E+09,9E+09,9E+09,9E+09,9E+09,9E+09]];
    CONST robtarget Target_7600:=[[191.595238644,60.131105214,27.024452337],[0.692516726,0.060687774,-0.040025666,0.717729422],[0,0,0,0],[9E+09,9E+09,9E+09,9E+09,9E+09,9E+09]];
    CONST robtarget Target_7610:=[[191.303557827,60.10058681,27.032171073],[0.692516726,0.060687774,-0.040025667,0.717729422],[0,0,0,0],[9E+09,9E+09,9E+09,9E+09,9E+09,9E+09]];
    CONST robtarget Target_7620:=[[190.055925774,60.053579659,27.065392638],[0.692516726,0.060687774,-0.040025667,0.717729422],[0,0,0,0],[9E+09,9E+09,9E+09,9E+09,9E+09,9E+09]];
    CONST robtarget Target_7630:=[[190.57270134,46.304002973,27.017752736],[0.692516726,0.060687774,-0.040025667,0.717729422],[0,0,0,0],[9E+09,9E+09,9E+09,9E+09,9E+09,9E+09]];
    CONST robtarget Target_7640:=[[190.564201274,46.010751964,27.017258304],[0.692516726,0.060687774,-0.040025667,0.717729422],[0,0,0,0],[9E+09,9E+09,9E+09,9E+09,9E+09,9E+09]];
    CONST robtarget Target_7650:=[[190.515246815,45.755034183,27.017937182],[0.692516726,0.060687774,-0.040025666,0.717729422],[0,0,0,0],[9E+09,9E+09,9E+09,9E+09,9E+09,9E+09]];
    CONST robtarget Target_7660:=[[190.425837963,45.536849632,27.019789369],[0.692516726,0.060687774,-0.040025667,0.717729422],[0,0,0,0],[9E+09,9E+09,9E+09,9E+09,9E+09,9E+09]];
    CONST robtarget Target_7670:=[[190.295974718,45.35619831,27.022814867],[0.692516726,0.060687774,-0.040025666,0.717729422],[0,0,0,0],[9E+09,9E+09,9E+09,9E+09,9E+09,9E+09]];
    CONST robtarget Target_7680:=[[190.125657081,45.213080218,27.027013674],[0.692516726,0.060687774,-0.040025667,0.717729422],[0,0,0,0],[9E+09,9E+09,9E+09,9E+09,9E+09,9E+09]];
    CONST robtarget Target_7690:=[[189.91488505,45.107495357,27.03238579],[0.692516726,0.060687774,-0.040025667,0.717729422],[0,0,0,0],[9E+09,9E+09,9E+09,9E+09,9E+09,9E+09]];
    CONST robtarget Target_7700:=[[189.663658627,45.039443724,27.038931217],[0.692516726,0.060687774,-0.040025666,0.717729422],[0,0,0,0],[9E+09,9E+09,9E+09,9E+09,9E+09,9E+09]];
    CONST robtarget Target_7710:=[[189.37197781,45.008925322,27.046649953],[0.692516726,0.060687774,-0.040025667,0.717729422],[0,0,0,0],[9E+09,9E+09,9E+09,9E+09,9E+09,9E+09]];
    CONST robtarget Target_7720:=[[189.078831101,45.017409122,27.054503826],[0.692516726,0.060687774,-0.040025666,0.717729422],[0,0,0,0],[9E+09,9E+09,9E+09,9E+09,9E+09,9E+09]];
    CONST robtarget Target_7730:=[[188.823207004,45.066364099,27.06145466],[0.692516726,0.060687774,-0.040025666,0.717729422],[0,0,0,0],[9E+09,9E+09,9E+09,9E+09,9E+09,9E+09]];
    CONST robtarget Target_7740:=[[188.605105516,45.155790252,27.067502456],[0.692516726,0.060687774,-0.040025666,0.717729422],[0,0,0,0],[9E+09,9E+09,9E+09,9E+09,9E+09,9E+09]];
    CONST robtarget Target_7750:=[[188.424526638,45.285687583,27.072647214],[0.692516726,0.060687774,-0.040025667,0.717729422],[0,0,0,0],[9E+09,9E+09,9E+09,9E+09,9E+09,9E+09]];
    CONST robtarget Target_7760:=[[188.281470372,45.456056091,27.076888934],[0.692516726,0.060687774,-0.040025666,0.717729422],[0,0,0,0],[9E+09,9E+09,9E+09,9E+09,9E+09,9E+09]];
    CONST robtarget Target_7770:=[[188.175936715,45.666895774,27.080227616],[0.692516726,0.060687774,-0.040025666,0.717729422],[0,0,0,0],[9E+09,9E+09,9E+09,9E+09,9E+09,9E+09]];
    CONST robtarget Target_7780:=[[188.107925669,45.918206634,27.08266326],[0.692516726,0.060687774,-0.040025667,0.717729422],[0,0,0,0],[9E+09,9E+09,9E+09,9E+09,9E+09,9E+09]];
    CONST robtarget Target_7790:=[[188.077437233,46.209988671,27.084195866],[0.692516726,0.060687774,-0.040025667,0.717729422],[0,0,0,0],[9E+09,9E+09,9E+09,9E+09,9E+09,9E+09]];
    CONST robtarget Target_7800:=[[187.560661667,59.959565356,27.131835768],[0.692516726,0.060687774,-0.040025667,0.717729422],[0,0,0,0],[9E+09,9E+09,9E+09,9E+09,9E+09,9E+09]];
    CONST robtarget Target_7810:=[[183.817765507,59.818543902,27.231500463],[0.692516726,0.060687774,-0.040025667,0.717729422],[0,0,0,0],[9E+09,9E+09,9E+09,9E+09,9E+09,9E+09]];
    CONST robtarget Target_7820:=[[183.5246188,59.827027703,27.239354335],[0.692516726,0.060687774,-0.040025666,0.717729422],[0,0,0,0],[9E+09,9E+09,9E+09,9E+09,9E+09,9E+09]];
    CONST robtarget Target_7830:=[[183.268994701,59.875982681,27.246305169],[0.692516726,0.060687774,-0.040025666,0.717729422],[0,0,0,0],[9E+09,9E+09,9E+09,9E+09,9E+09,9E+09]];
    CONST robtarget Target_7840:=[[183.050893214,59.965408834,27.252352965],[0.692516726,0.060687774,-0.040025666,0.717729422],[0,0,0,0],[9E+09,9E+09,9E+09,9E+09,9E+09,9E+09]];
    CONST robtarget Target_7850:=[[182.870314337,60.095306165,27.257497723],[0.692516726,0.060687774,-0.040025667,0.717729422],[0,0,0,0],[9E+09,9E+09,9E+09,9E+09,9E+09,9E+09]];
    CONST robtarget Target_7860:=[[182.72725807,60.265674671,27.261739444],[0.692516726,0.060687774,-0.040025666,0.717729422],[0,0,0,0],[9E+09,9E+09,9E+09,9E+09,9E+09,9E+09]];
    CONST robtarget Target_7870:=[[182.621724413,60.476514355,27.265078126],[0.692516726,0.060687774,-0.040025666,0.717729422],[0,0,0,0],[9E+09,9E+09,9E+09,9E+09,9E+09,9E+09]];
    CONST robtarget Target_7880:=[[182.553713367,60.727825215,27.26751377],[0.692516726,0.060687774,-0.040025667,0.717729422],[0,0,0,0],[9E+09,9E+09,9E+09,9E+09,9E+09,9E+09]];
    CONST robtarget Target_7890:=[[182.523224931,61.019607252,27.269046376],[0.692516726,0.060687774,-0.040025667,0.717729422],[0,0,0,0],[9E+09,9E+09,9E+09,9E+09,9E+09,9E+09]];
    CONST robtarget Target_7900:=[[182.531724996,61.312858263,27.269540808],[0.692516726,0.060687774,-0.040025667,0.717729422],[0,0,0,0],[9E+09,9E+09,9E+09,9E+09,9E+09,9E+09]];
    CONST robtarget Target_7910:=[[182.580679456,61.568576043,27.26886193],[0.692516726,0.060687774,-0.040025666,0.717729422],[0,0,0,0],[9E+09,9E+09,9E+09,9E+09,9E+09,9E+09]];
    CONST robtarget Target_7920:=[[182.670088307,61.786760594,27.267009743],[0.692516726,0.060687774,-0.040025667,0.717729422],[0,0,0,0],[9E+09,9E+09,9E+09,9E+09,9E+09,9E+09]];
    CONST robtarget Target_7930:=[[182.799951552,61.967411916,27.263984246],[0.692516726,0.060687774,-0.040025666,0.717729422],[0,0,0,0],[9E+09,9E+09,9E+09,9E+09,9E+09,9E+09]];
    CONST robtarget Target_7940:=[[182.970269189,62.110530007,27.259785439],[0.692516726,0.060687774,-0.040025667,0.717729422],[0,0,0,0],[9E+09,9E+09,9E+09,9E+09,9E+09,9E+09]];
    CONST robtarget Target_7950:=[[183.18104122,62.21611487,27.254413322],[0.692516726,0.060687774,-0.040025667,0.717729422],[0,0,0,0],[9E+09,9E+09,9E+09,9E+09,9E+09,9E+09]];
    CONST robtarget Target_7960:=[[183.432267644,62.284166502,27.247867895],[0.692516726,0.060687774,-0.040025666,0.717729422],[0,0,0,0],[9E+09,9E+09,9E+09,9E+09,9E+09,9E+09]];
    CONST robtarget Target_7970:=[[183.72394846,62.314684905,27.240149159],[0.692516726,0.060687774,-0.040025667,0.717729422],[0,0,0,0],[9E+09,9E+09,9E+09,9E+09,9E+09,9E+09]];
    CONST robtarget Target_7980:=[[187.46684462,62.455706359,27.140484464],[0.692516726,0.060687774,-0.040025667,0.717729422],[0,0,0,0],[9E+09,9E+09,9E+09,9E+09,9E+09,9E+09]];
    CONST robtarget Target_7990:=[[187.232302003,68.696058863,27.162106205],[0.692516726,0.060687774,-0.040025667,0.717729422],[0,0,0,0],[9E+09,9E+09,9E+09,9E+09,9E+09,9E+09]];
    CONST robtarget Target_8000:=[[186.430978427,68.769848651,-2.827099113],[0.692516726,0.060687774,-0.040025667,0.717729422],[0,0,0,0],[9E+09,9E+09,9E+09,9E+09,9E+09,9E+09]];
    CONST robtarget Target_8010:=[[174.147612776,62.057857728,-2.515397819],[0.692516726,0.060687774,-0.040025667,0.717729422],[0,0,0,0],[9E+09,9E+09,9E+09,9E+09,9E+09,9E+09]];
    CONST robtarget Target_8020:=[[174.948936353,61.98406794,27.473807499],[0.692516726,0.060687774,-0.040025667,0.717729422],[0,0,0,0],[9E+09,9E+09,9E+09,9E+09,9E+09,9E+09]];
    CONST robtarget Target_8030:=[[169.95840814,61.796039335,27.606693759],[0.692516726,0.060687774,-0.040025667,0.717729422],[0,0,0,0],[9E+09,9E+09,9E+09,9E+09,9E+09,9E+09]];
    CONST robtarget Target_8040:=[[169.444446461,61.754053988,27.620323714],[0.692516726,0.060687774,-0.040025667,0.717729422],[0,0,0,0],[9E+09,9E+09,9E+09,9E+09,9E+09,9E+09]];
    CONST robtarget Target_8050:=[[168.952651737,61.667662301,27.633252095],[0.692516726,0.060687774,-0.040025667,0.717729422],[0,0,0,0],[9E+09,9E+09,9E+09,9E+09,9E+09,9E+09]];
    CONST robtarget Target_8060:=[[168.483023967,61.536864272,27.645478903],[0.692516726,0.060687774,-0.040025667,0.717729422],[0,0,0,0],[9E+09,9E+09,9E+09,9E+09,9E+09,9E+09]];
    CONST robtarget Target_8070:=[[168.03556315,61.361659902,27.657004137],[0.692516726,0.060687774,-0.040025667,0.717729422],[0,0,0,0],[9E+09,9E+09,9E+09,9E+09,9E+09,9E+09]];
    CONST robtarget Target_8080:=[[167.610269289,61.142049192,27.667827797],[0.692516726,0.060687774,-0.040025667,0.717729422],[0,0,0,0],[9E+09,9E+09,9E+09,9E+09,9E+09,9E+09]];
    CONST robtarget Target_8090:=[[167.207142381,60.878032142,27.677949884],[0.692516726,0.060687774,-0.040025666,0.717729422],[0,0,0,0],[9E+09,9E+09,9E+09,9E+09,9E+09,9E+09]];
    CONST robtarget Target_8100:=[[166.826182427,60.569608749,27.687370397],[0.692516726,0.060687774,-0.040025666,0.717729422],[0,0,0,0],[9E+09,9E+09,9E+09,9E+09,9E+09,9E+09]];
    CONST robtarget Target_8110:=[[166.467389428,60.216779016,27.696089336],[0.692516726,0.060687774,-0.040025666,0.717729422],[0,0,0,0],[9E+09,9E+09,9E+09,9E+09,9E+09,9E+09]];
    CONST robtarget Target_8120:=[[166.142645543,59.832358815,27.703820739],[0.692516726,0.060687774,-0.040025666,0.717729422],[0,0,0,0],[9E+09,9E+09,9E+09,9E+09,9E+09,9E+09]];
    CONST robtarget Target_8130:=[[165.863832932,59.429164018,27.710278645],[0.692516726,0.060687774,-0.040025667,0.717729422],[0,0,0,0],[9E+09,9E+09,9E+09,9E+09,9E+09,9E+09]];
    CONST robtarget Target_8140:=[[165.630951595,59.007194625,27.715463053],[0.692516726,0.060687774,-0.040025666,0.717729422],[0,0,0,0],[9E+09,9E+09,9E+09,9E+09,9E+09,9E+09]];
    CONST robtarget Target_8150:=[[165.444001531,58.566450637,27.719373963],[0.692516726,0.060687774,-0.040025666,0.717729422],[0,0,0,0],[9E+09,9E+09,9E+09,9E+09,9E+09,9E+09]];
    CONST robtarget Target_8160:=[[165.302982743,58.106932052,27.722011376],[0.692516726,0.060687774,-0.040025666,0.717729422],[0,0,0,0],[9E+09,9E+09,9E+09,9E+09,9E+09,9E+09]];
    CONST robtarget Target_8170:=[[165.207895228,57.628638873,27.72337529],[0.692516726,0.060687774,-0.040025667,0.717729422],[0,0,0,0],[9E+09,9E+09,9E+09,9E+09,9E+09,9E+09]];
    CONST robtarget Target_8180:=[[165.158738987,57.131571097,27.723465707],[0.692516726,0.060687774,-0.040025666,0.717729422],[0,0,0,0],[9E+09,9E+09,9E+09,9E+09,9E+09,9E+09]];
    CONST robtarget Target_8190:=[[165.155514021,56.615728725,27.722282626],[0.692516726,0.060687774,-0.040025667,0.717729422],[0,0,0,0],[9E+09,9E+09,9E+09,9E+09,9E+09,9E+09]];
    CONST robtarget Target_8200:=[[165.57847254,45.362293041,27.683291421],[0.692516726,0.060687774,-0.040025667,0.717729422],[0,0,0,0],[9E+09,9E+09,9E+09,9E+09,9E+09,9E+09]];
    CONST robtarget Target_8210:=[[165.608960975,45.070511005,27.681758815],[0.692516726,0.060687774,-0.040025667,0.717729422],[0,0,0,0],[9E+09,9E+09,9E+09,9E+09,9E+09,9E+09]];
    CONST robtarget Target_8220:=[[165.676972022,44.819200145,27.679323171],[0.692516726,0.060687774,-0.040025666,0.717729422],[0,0,0,0],[9E+09,9E+09,9E+09,9E+09,9E+09,9E+09]];
    CONST robtarget Target_8230:=[[165.782505679,44.608360461,27.675984488],[0.692516726,0.060687774,-0.040025666,0.717729422],[0,0,0,0],[9E+09,9E+09,9E+09,9E+09,9E+09,9E+09]];
    CONST robtarget Target_8240:=[[165.925561945,44.437991954,27.671742768],[0.692516726,0.060687774,-0.040025667,0.717729422],[0,0,0,0],[9E+09,9E+09,9E+09,9E+09,9E+09,9E+09]];
    CONST robtarget Target_8250:=[[166.106140823,44.308094623,27.66659801],[0.692516726,0.060687774,-0.040025666,0.717729422],[0,0,0,0],[9E+09,9E+09,9E+09,9E+09,9E+09,9E+09]];
    CONST robtarget Target_8260:=[[166.32424231,44.21866847,27.660550214],[0.692516726,0.060687774,-0.040025666,0.717729422],[0,0,0,0],[9E+09,9E+09,9E+09,9E+09,9E+09,9E+09]];
    CONST robtarget Target_8270:=[[166.579866408,44.169713492,27.65359938],[0.692516726,0.060687774,-0.040025666,0.717729422],[0,0,0,0],[9E+09,9E+09,9E+09,9E+09,9E+09,9E+09]];
    CONST robtarget Target_8280:=[[166.873013116,44.161229692,27.645745508],[0.692516726,0.060687774,-0.040025667,0.717729422],[0,0,0,0],[9E+09,9E+09,9E+09,9E+09,9E+09,9E+09]];
    CONST robtarget Target_8290:=[[173.111173382,44.396265449,27.479637683],[0.692516726,0.060687774,-0.040025667,0.717729422],[0,0,0,0],[9E+09,9E+09,9E+09,9E+09,9E+09,9E+09]];
    CONST robtarget Target_8300:=[[173.625135061,44.438250795,27.466007728],[0.692516726,0.060687774,-0.040025667,0.717729422],[0,0,0,0],[9E+09,9E+09,9E+09,9E+09,9E+09,9E+09]];
    CONST robtarget Target_8310:=[[174.116929785,44.524642483,27.453079347],[0.692516726,0.060687774,-0.040025667,0.717729422],[0,0,0,0],[9E+09,9E+09,9E+09,9E+09,9E+09,9E+09]];
    CONST robtarget Target_8320:=[[174.586557556,44.655440512,27.440852539],[0.692516726,0.060687774,-0.040025667,0.717729422],[0,0,0,0],[9E+09,9E+09,9E+09,9E+09,9E+09,9E+09]];
    CONST robtarget Target_8330:=[[175.034018371,44.830644881,27.429327305],[0.692516726,0.060687774,-0.040025667,0.717729422],[0,0,0,0],[9E+09,9E+09,9E+09,9E+09,9E+09,9E+09]];
    CONST robtarget Target_8340:=[[175.459312234,45.050255591,27.418503645],[0.692516726,0.060687774,-0.040025667,0.717729422],[0,0,0,0],[9E+09,9E+09,9E+09,9E+09,9E+09,9E+09]];
    CONST robtarget Target_8350:=[[175.862439142,45.314272643,27.408381558],[0.692516726,0.060687774,-0.040025666,0.717729422],[0,0,0,0],[9E+09,9E+09,9E+09,9E+09,9E+09,9E+09]];
    CONST robtarget Target_8360:=[[176.243399095,45.622696035,27.398961045],[0.692516726,0.060687774,-0.040025666,0.717729422],[0,0,0,0],[9E+09,9E+09,9E+09,9E+09,9E+09,9E+09]];
    CONST robtarget Target_8370:=[[176.602192094,45.975525768,27.390242106],[0.692516726,0.060687774,-0.040025666,0.717729422],[0,0,0,0],[9E+09,9E+09,9E+09,9E+09,9E+09,9E+09]];
    CONST robtarget Target_8380:=[[176.926935979,46.359945969,27.382510702],[0.692516726,0.060687774,-0.040025666,0.717729422],[0,0,0,0],[9E+09,9E+09,9E+09,9E+09,9E+09,9E+09]];
    CONST robtarget Target_8390:=[[177.20574859,46.763140766,27.376052797],[0.692516726,0.060687774,-0.040025667,0.717729422],[0,0,0,0],[9E+09,9E+09,9E+09,9E+09,9E+09,9E+09]];
    CONST robtarget Target_8400:=[[177.438629927,47.185110158,27.370868389],[0.692516726,0.060687774,-0.040025666,0.717729422],[0,0,0,0],[9E+09,9E+09,9E+09,9E+09,9E+09,9E+09]];
    CONST robtarget Target_8410:=[[177.62557999,47.625854147,27.366957479],[0.692516726,0.060687774,-0.040025666,0.717729422],[0,0,0,0],[9E+09,9E+09,9E+09,9E+09,9E+09,9E+09]];
    CONST robtarget Target_8420:=[[177.766598779,48.085372732,27.364320066],[0.692516726,0.060687774,-0.040025666,0.717729422],[0,0,0,0],[9E+09,9E+09,9E+09,9E+09,9E+09,9E+09]];
    CONST robtarget Target_8430:=[[177.861686294,48.563665911,27.362956152],[0.692516726,0.060687774,-0.040025667,0.717729422],[0,0,0,0],[9E+09,9E+09,9E+09,9E+09,9E+09,9E+09]];
    CONST robtarget Target_8440:=[[177.910842535,49.060733687,27.362865735],[0.692516726,0.060687774,-0.040025666,0.717729422],[0,0,0,0],[9E+09,9E+09,9E+09,9E+09,9E+09,9E+09]];
    CONST robtarget Target_8450:=[[177.914067502,49.576576058,27.364048816],[0.692516726,0.060687774,-0.040025667,0.717729422],[0,0,0,0],[9E+09,9E+09,9E+09,9E+09,9E+09,9E+09]];
    CONST robtarget Target_8460:=[[177.891401022,49.911290502,27.365478053],[0.692516726,0.060687774,-0.040025667,0.717729422],[0,0,0,0],[9E+09,9E+09,9E+09,9E+09,9E+09,9E+09]];
    CONST robtarget Target_8470:=[[177.848810367,50.239395646,27.36742341],[0.692516726,0.060687774,-0.040025666,0.717729422],[0,0,0,0],[9E+09,9E+09,9E+09,9E+09,9E+09,9E+09]];
    CONST robtarget Target_8480:=[[177.786295537,50.56089149,27.369884886],[0.692516726,0.060687774,-0.040025666,0.717729422],[0,0,0,0],[9E+09,9E+09,9E+09,9E+09,9E+09,9E+09]];
    CONST robtarget Target_8490:=[[177.703856531,50.875778034,27.372862482],[0.692516726,0.060687774,-0.040025666,0.717729422],[0,0,0,0],[9E+09,9E+09,9E+09,9E+09,9E+09,9E+09]];
    CONST robtarget Target_8500:=[[177.601493349,51.184055277,27.376356197],[0.692516726,0.060687774,-0.040025667,0.717729422],[0,0,0,0],[9E+09,9E+09,9E+09,9E+09,9E+09,9E+09]];
    CONST robtarget Target_8510:=[[177.479205993,51.48572322,27.380366032],[0.692516726,0.060687774,-0.040025667,0.717729422],[0,0,0,0],[9E+09,9E+09,9E+09,9E+09,9E+09,9E+09]];
    CONST robtarget Target_8520:=[[177.33699446,51.780781864,27.384891986],[0.692516726,0.060687774,-0.040025667,0.717729422],[0,0,0,0],[9E+09,9E+09,9E+09,9E+09,9E+09,9E+09]];
    CONST robtarget Target_8530:=[[177.174858753,52.069231207,27.389934059],[0.692516726,0.060687774,-0.040025667,0.717729422],[0,0,0,0],[9E+09,9E+09,9E+09,9E+09,9E+09,9E+09]];
    CONST robtarget Target_8540:=[[176.97847861,52.362004826,27.395901798],[0.692516726,0.060687774,-0.040025666,0.717729422],[0,0,0,0],[9E+09,9E+09,9E+09,9E+09,9E+09,9E+09]];
    CONST robtarget Target_8550:=[[176.771291206,52.63500528,27.402109659],[0.692516726,0.060687774,-0.040025667,0.717729422],[0,0,0,0],[9E+09,9E+09,9E+09,9E+09,9E+09,9E+09]];
    CONST robtarget Target_8560:=[[176.553296542,52.888232571,27.40855764],[0.692516726,0.060687774,-0.040025667,0.717729422],[0,0,0,0],[9E+09,9E+09,9E+09,9E+09,9E+09,9E+09]];
    CONST robtarget Target_8570:=[[176.324494617,53.121686699,27.415245744],[0.692516726,0.060687774,-0.040025666,0.717729422],[0,0,0,0],[9E+09,9E+09,9E+09,9E+09,9E+09,9E+09]];
    CONST robtarget Target_8580:=[[176.084885432,53.335367662,27.422173969],[0.692516726,0.060687774,-0.040025667,0.717729422],[0,0,0,0],[9E+09,9E+09,9E+09,9E+09,9E+09,9E+09]];
    CONST robtarget Target_8590:=[[175.834468987,53.529275462,27.429342315],[0.692516726,0.060687774,-0.040025667,0.717729422],[0,0,0,0],[9E+09,9E+09,9E+09,9E+09,9E+09,9E+09]];
    CONST robtarget Target_8600:=[[175.57324528,53.703410098,27.436750784],[0.692516726,0.060687774,-0.040025667,0.717729422],[0,0,0,0],[9E+09,9E+09,9E+09,9E+09,9E+09,9E+09]];
    CONST robtarget Target_8610:=[[175.301214313,53.85777157,27.444399373],[0.692516726,0.060687774,-0.040025667,0.717729422],[0,0,0,0],[9E+09,9E+09,9E+09,9E+09,9E+09,9E+09]];
    CONST robtarget Target_8620:=[[175.018376086,53.99235988,27.452288085],[0.692516726,0.060687774,-0.040025667,0.717729422],[0,0,0,0],[9E+09,9E+09,9E+09,9E+09,9E+09,9E+09]];
    CONST robtarget Target_8630:=[[174.724730597,54.107175025,27.460416917],[0.692516726,0.060687774,-0.040025666,0.717729422],[0,0,0,0],[9E+09,9E+09,9E+09,9E+09,9E+09,9E+09]];
    CONST robtarget Target_8640:=[[174.420277849,54.202217005,27.468785872],[0.692516726,0.060687774,-0.040025666,0.717729422],[0,0,0,0],[9E+09,9E+09,9E+09,9E+09,9E+09,9E+09]];
    CONST robtarget Target_8650:=[[174.10501784,54.277485823,27.477394948],[0.692516726,0.060687774,-0.040025667,0.717729422],[0,0,0,0],[9E+09,9E+09,9E+09,9E+09,9E+09,9E+09]];
    CONST robtarget Target_8660:=[[173.778950569,54.332981477,27.486244146],[0.692516726,0.060687774,-0.040025666,0.717729422],[0,0,0,0],[9E+09,9E+09,9E+09,9E+09,9E+09,9E+09]];
    CONST robtarget Target_8670:=[[173.442076038,54.368703968,27.495333465],[0.692516726,0.060687774,-0.040025667,0.717729422],[0,0,0,0],[9E+09,9E+09,9E+09,9E+09,9E+09,9E+09]];
    CONST robtarget Target_8680:=[[173.094394247,54.384653294,27.504662905],[0.692516726,0.060687774,-0.040025667,0.717729422],[0,0,0,0],[9E+09,9E+09,9E+09,9E+09,9E+09,9E+09]];
    CONST robtarget Target_8690:=[[172.735905195,54.380829457,27.514232468],[0.692516726,0.060687774,-0.040025667,0.717729422],[0,0,0,0],[9E+09,9E+09,9E+09,9E+09,9E+09,9E+09]];
    CONST robtarget Target_8700:=[[167.745376982,54.192800851,27.647118727],[0.692516726,0.060687774,-0.040025667,0.717729422],[0,0,0,0],[9E+09,9E+09,9E+09,9E+09,9E+09,9E+09]];
    CONST robtarget Target_8710:=[[167.650778127,56.709743028,27.655839496],[0.692516726,0.060687774,-0.040025667,0.717729422],[0,0,0,0],[9E+09,9E+09,9E+09,9E+09,9E+09,9E+09]];
    CONST robtarget Target_8720:=[[166.84945455,56.783532816,-2.333365822],[0.692516726,0.060687774,-0.040025667,0.717729422],[0,0,0,0],[9E+09,9E+09,9E+09,9E+09,9E+09,9E+09]];
    CONST robtarget Target_8730:=[[102.509529144,132.906987315,-0.426872065],[0.692516726,0.060687774,-0.040025667,0.717729422],[0,0,0,0],[9E+09,9E+09,9E+09,9E+09,9E+09,9E+09]];
    CONST robtarget Target_8740:=[[103.310852721,132.833197528,29.562333253],[0.692516726,0.060687774,-0.040025667,0.717729422],[0,0,0,0],[9E+09,9E+09,9E+09,9E+09,9E+09,9E+09]];
    CONST robtarget Target_8750:=[[102.875041022,144.428611022,29.602509352],[0.692516726,0.060687774,-0.040025667,0.717729422],[0,0,0,0],[9E+09,9E+09,9E+09,9E+09,9E+09,9E+09]];
    CONST robtarget Target_8760:=[[92.885667049,144.05224043,29.868503349],[0.692516726,0.060687774,-0.040025667,0.717729422],[0,0,0,0],[9E+09,9E+09,9E+09,9E+09,9E+09,9E+09]];
    CONST robtarget Target_8770:=[[93.321478748,132.456826936,29.82832725],[0.692516726,0.060687774,-0.040025667,0.717729422],[0,0,0,0],[9E+09,9E+09,9E+09,9E+09,9E+09,9E+09]];
    CONST robtarget Target_8780:=[[71.344856007,131.628811634,30.413514042],[0.692516726,0.060687774,-0.040025667,0.717729422],[0,0,0,0],[9E+09,9E+09,9E+09,9E+09,9E+09,9E+09]];
    CONST robtarget Target_8790:=[[70.562998931,131.560804242,30.434238241],[0.692516726,0.060687774,-0.040025667,0.717729422],[0,0,0,0],[9E+09,9E+09,9E+09,9E+09,9E+09,9E+09]];
    CONST robtarget Target_8800:=[[69.791565205,131.416462247,30.454496099],[0.692516726,0.060687774,-0.040025666,0.717729422],[0,0,0,0],[9E+09,9E+09,9E+09,9E+09,9E+09,9E+09]];
    CONST robtarget Target_8810:=[[69.037984158,131.19717574,30.474092522],[0.692516726,0.060687774,-0.040025667,0.717729422],[0,0,0,0],[9E+09,9E+09,9E+09,9E+09,9E+09,9E+09]];
    CONST robtarget Target_8820:=[[68.309513187,130.905056571,30.492838786],[0.692516726,0.060687774,-0.040025666,0.717729422],[0,0,0,0],[9E+09,9E+09,9E+09,9E+09,9E+09,9E+09]];
    CONST robtarget Target_8830:=[[67.613167868,130.542918006,30.510554353],[0.692516726,0.060687774,-0.040025667,0.717729422],[0,0,0,0],[9E+09,9E+09,9E+09,9E+09,9E+09,9E+09]];
    CONST robtarget Target_8840:=[[66.955654384,130.114247639,30.527068614],[0.692516726,0.060687774,-0.040025666,0.717729422],[0,0,0,0],[9E+09,9E+09,9E+09,9E+09,9E+09,9E+09]];
    CONST robtarget Target_8850:=[[66.343304951,129.623173799,30.542222527],[0.692516726,0.060687774,-0.040025667,0.717729422],[0,0,0,0],[9E+09,9E+09,9E+09,9E+09,9E+09,9E+09]];
    CONST robtarget Target_8860:=[[65.782016828,129.074425795,30.555870152],[0.692516726,0.060687774,-0.040025666,0.717729422],[0,0,0,0],[9E+09,9E+09,9E+09,9E+09,9E+09,9E+09]];
    CONST robtarget Target_8870:=[[65.277195527,128.473288372,30.567880053],[0.692516726,0.060687774,-0.040025667,0.717729422],[0,0,0,0],[9E+09,9E+09,9E+09,9E+09,9E+09,9E+09]];
    CONST robtarget Target_8880:=[[64.833702753,127.82555081,30.57813657],[0.692516726,0.060687774,-0.040025667,0.717729422],[0,0,0,0],[9E+09,9E+09,9E+09,9E+09,9E+09,9E+09]];
    CONST robtarget Target_8890:=[[64.455809583,127.137451176,30.586540927],[0.692516726,0.060687774,-0.040025666,0.717729422],[0,0,0,0],[9E+09,9E+09,9E+09,9E+09,9E+09,9E+09]];
    CONST robtarget Target_8900:=[[64.147155337,126.415616247,30.593012185],[0.692516726,0.060687774,-0.040025667,0.717729422],[0,0,0,0],[9E+09,9E+09,9E+09,9E+09,9E+09,9E+09]];
    CONST robtarget Target_8910:=[[63.910712522,125.666997688,30.597488022],[0.692516726,0.060687774,-0.040025667,0.717729422],[0,0,0,0],[9E+09,9E+09,9E+09,9E+09,9E+09,9E+09]];
    CONST robtarget Target_8920:=[[63.748758213,124.898805103,30.599925334],[0.692516726,0.060687774,-0.040025667,0.717729422],[0,0,0,0],[9E+09,9E+09,9E+09,9E+09,9E+09,9E+09]];
    CONST robtarget Target_8930:=[[63.662852117,124.118436608,30.600300647],[0.692516726,0.060687774,-0.040025667,0.717729422],[0,0,0,0],[9E+09,9E+09,9E+09,9E+09,9E+09,9E+09]];
    CONST robtarget Target_8940:=[[63.653821557,123.333407578,30.598610348],[0.692516726,0.060687774,-0.040025667,0.717729422],[0,0,0,0],[9E+09,9E+09,9E+09,9E+09,9E+09,9E+09]];
    CONST robtarget Target_8950:=[[64.300665588,106.123167381,30.538979847],[0.692516726,0.060687774,-0.040025667,0.717729422],[0,0,0,0],[9E+09,9E+09,9E+09,9E+09,9E+09,9E+09]];
    CONST robtarget Target_8960:=[[63.518808512,106.055159989,30.559704046],[0.692516726,0.060687774,-0.040025667,0.717729422],[0,0,0,0],[9E+09,9E+09,9E+09,9E+09,9E+09,9E+09]];
    CONST robtarget Target_8970:=[[62.747374786,105.910817994,30.579961904],[0.692516726,0.060687774,-0.040025666,0.717729422],[0,0,0,0],[9E+09,9E+09,9E+09,9E+09,9E+09,9E+09]];
    CONST robtarget Target_8980:=[[61.993793739,105.691531488,30.599558327],[0.692516726,0.060687774,-0.040025667,0.717729422],[0,0,0,0],[9E+09,9E+09,9E+09,9E+09,9E+09,9E+09]];
    CONST robtarget Target_8990:=[[61.265322769,105.399412319,30.618304591],[0.692516726,0.060687774,-0.040025666,0.717729422],[0,0,0,0],[9E+09,9E+09,9E+09,9E+09,9E+09,9E+09]];
    CONST robtarget Target_9000:=[[60.568977449,105.037273754,30.636020158],[0.692516726,0.060687774,-0.040025667,0.717729422],[0,0,0,0],[9E+09,9E+09,9E+09,9E+09,9E+09,9E+09]];
    CONST robtarget Target_9010:=[[59.911463965,104.608603386,30.652534419],[0.692516726,0.060687774,-0.040025666,0.717729422],[0,0,0,0],[9E+09,9E+09,9E+09,9E+09,9E+09,9E+09]];
    CONST robtarget Target_9020:=[[59.299114532,104.117529547,30.667688332],[0.692516726,0.060687774,-0.040025667,0.717729422],[0,0,0,0],[9E+09,9E+09,9E+09,9E+09,9E+09,9E+09]];
    CONST robtarget Target_9030:=[[58.737826409,103.568781543,30.681335957],[0.692516726,0.060687774,-0.040025666,0.717729422],[0,0,0,0],[9E+09,9E+09,9E+09,9E+09,9E+09,9E+09]];
    CONST robtarget Target_9040:=[[58.233005108,102.967644119,30.693345858],[0.692516726,0.060687774,-0.040025667,0.717729422],[0,0,0,0],[9E+09,9E+09,9E+09,9E+09,9E+09,9E+09]];
    CONST robtarget Target_9050:=[[57.789512335,102.319906557,30.703602375],[0.692516726,0.060687774,-0.040025667,0.717729422],[0,0,0,0],[9E+09,9E+09,9E+09,9E+09,9E+09,9E+09]];
    CONST robtarget Target_9060:=[[57.411619165,101.631806924,30.712006732],[0.692516726,0.060687774,-0.040025666,0.717729422],[0,0,0,0],[9E+09,9E+09,9E+09,9E+09,9E+09,9E+09]];
    CONST robtarget Target_9070:=[[57.102964918,100.909971995,30.71847799],[0.692516726,0.060687774,-0.040025667,0.717729422],[0,0,0,0],[9E+09,9E+09,9E+09,9E+09,9E+09,9E+09]];
    CONST robtarget Target_9080:=[[56.866522103,100.161353435,30.722953827],[0.692516726,0.060687774,-0.040025667,0.717729422],[0,0,0,0],[9E+09,9E+09,9E+09,9E+09,9E+09,9E+09]];
    CONST robtarget Target_9090:=[[56.704567794,99.39316085,30.725391139],[0.692516726,0.060687774,-0.040025667,0.717729422],[0,0,0,0],[9E+09,9E+09,9E+09,9E+09,9E+09,9E+09]];
    CONST robtarget Target_9100:=[[56.618661698,98.612792356,30.725766452],[0.692516726,0.060687774,-0.040025667,0.717729422],[0,0,0,0],[9E+09,9E+09,9E+09,9E+09,9E+09,9E+09]];
    CONST robtarget Target_9110:=[[56.609631138,97.827763325,30.724076153],[0.692516726,0.060687774,-0.040025667,0.717729422],[0,0,0,0],[9E+09,9E+09,9E+09,9E+09,9E+09,9E+09]];
    CONST robtarget Target_9120:=[[56.677563085,97.045634019,30.72033652],[0.692516726,0.060687774,-0.040025667,0.717729422],[0,0,0,0],[9E+09,9E+09,9E+09,9E+09,9E+09,9E+09]];
    CONST robtarget Target_9130:=[[56.821803315,96.273936769,30.714583567],[0.692516726,0.060687774,-0.040025667,0.717729422],[0,0,0,0],[9E+09,9E+09,9E+09,9E+09,9E+09,9E+09]];
    CONST robtarget Target_9140:=[[57.040962717,95.520103442,30.7068727],[0.692516726,0.060687774,-0.040025666,0.717729422],[0,0,0,0],[9E+09,9E+09,9E+09,9E+09,9E+09,9E+09]];
    CONST robtarget Target_9150:=[[57.332930665,94.791393865,30.697278177],[0.692516726,0.060687774,-0.040025666,0.717729422],[0,0,0,0],[9E+09,9E+09,9E+09,9E+09,9E+09,9E+09]];
    CONST robtarget Target_9160:=[[57.69489535,94.094825908,30.685892398],[0.692516726,0.060687774,-0.040025667,0.717729422],[0,0,0,0],[9E+09,9E+09,9E+09,9E+09,9E+09,9E+09]];
    CONST robtarget Target_9170:=[[58.123370853,93.437107905,30.672825017],[0.692516726,0.060687774,-0.040025667,0.717729422],[0,0,0,0],[9E+09,9E+09,9E+09,9E+09,9E+09,9E+09]];
    CONST robtarget Target_9180:=[[58.61423072,92.824574036,30.658201877],[0.692516726,0.060687774,-0.040025667,0.717729422],[0,0,0,0],[9E+09,9E+09,9E+09,9E+09,9E+09,9E+09]];
    CONST robtarget Target_9190:=[[59.162747703,92.263123339,30.642163809],[0.692516726,0.060687774,-0.040025667,0.717729422],[0,0,0,0],[9E+09,9E+09,9E+09,9E+09,9E+09,9E+09]];
    CONST robtarget Target_9200:=[[59.763639284,91.75816289,30.624865268],[0.692516726,0.060687774,-0.040025666,0.717729422],[0,0,0,0],[9E+09,9E+09,9E+09,9E+09,9E+09,9E+09]];
    CONST robtarget Target_9210:=[[60.411118547,91.314555735,30.606472847],[0.692516726,0.060687774,-0.040025667,0.717729422],[0,0,0,0],[9E+09,9E+09,9E+09,9E+09,9E+09,9E+09]];
    CONST robtarget Target_9220:=[[61.098949915,90.936574053,30.587163676],[0.692516726,0.060687774,-0.040025667,0.717729422],[0,0,0,0],[9E+09,9E+09,9E+09,9E+09,9E+09,9E+09]];
    CONST robtarget Target_9230:=[[61.820509194,90.627858015,30.567123714],[0.692516726,0.060687774,-0.040025667,0.717729422],[0,0,0,0],[9E+09,9E+09,9E+09,9E+09,9E+09,9E+09]];
    CONST robtarget Target_9240:=[[62.568847375,90.391380724,30.546545955],[0.692516726,0.060687774,-0.040025666,0.717729422],[0,0,0,0],[9E+09,9E+09,9E+09,9E+09,9E+09,9E+09]];
    CONST robtarget Target_9250:=[[63.336757552,90.229419587,30.525628575],[0.692516726,0.060687774,-0.040025667,0.717729422],[0,0,0,0],[9E+09,9E+09,9E+09,9E+09,9E+09,9E+09]];
    CONST robtarget Target_9260:=[[64.11684433,90.143534378,30.504573019],[0.692516726,0.060687774,-0.040025666,0.717729422],[0,0,0,0],[9E+09,9E+09,9E+09,9E+09,9E+09,9E+09]];
    CONST robtarget Target_9270:=[[64.901595045,90.134552217,30.483582065],[0.692516726,0.060687774,-0.040025667,0.717729422],[0,0,0,0],[9E+09,9E+09,9E+09,9E+09,9E+09,9E+09]];
    CONST robtarget Target_9280:=[[65.681958473,69.371831399,30.411642834],[0.692516726,0.060687774,-0.040025666,0.717729422],[0,0,0,0],[9E+09,9E+09,9E+09,9E+09,9E+09,9E+09]];
    CONST robtarget Target_9290:=[[65.74989042,68.589702092,30.4079032],[0.692516726,0.060687774,-0.040025666,0.717729422],[0,0,0,0],[9E+09,9E+09,9E+09,9E+09,9E+09,9E+09]];
    CONST robtarget Target_9300:=[[65.89413065,67.818004842,30.402150248],[0.692516726,0.060687774,-0.040025666,0.717729422],[0,0,0,0],[9E+09,9E+09,9E+09,9E+09,9E+09,9E+09]];
    CONST robtarget Target_9310:=[[66.113290051,67.064171514,30.39443938],[0.692516727,0.060687774,-0.040025666,0.717729422],[0,0,0,0],[9E+09,9E+09,9E+09,9E+09,9E+09,9E+09]];
    CONST robtarget Target_9320:=[[66.405258,66.335461938,30.384844857],[0.692516727,0.060687774,-0.040025666,0.717729422],[0,0,0,0],[9E+09,9E+09,9E+09,9E+09,9E+09,9E+09]];
    CONST robtarget Target_9330:=[[66.767222684,65.638893982,30.373459079],[0.692516726,0.060687774,-0.040025666,0.717729422],[0,0,0,0],[9E+09,9E+09,9E+09,9E+09,9E+09,9E+09]];
    CONST robtarget Target_9340:=[[67.195698187,64.981175977,30.360391697],[0.692516726,0.060687774,-0.040025666,0.717729422],[0,0,0,0],[9E+09,9E+09,9E+09,9E+09,9E+09,9E+09]];
    CONST robtarget Target_9350:=[[67.686558054,64.368642108,30.345768558],[0.692516726,0.060687774,-0.040025666,0.717729422],[0,0,0,0],[9E+09,9E+09,9E+09,9E+09,9E+09,9E+09]];
    CONST robtarget Target_9360:=[[68.235075038,63.807191411,30.32973049],[0.692516726,0.060687774,-0.040025666,0.717729422],[0,0,0,0],[9E+09,9E+09,9E+09,9E+09,9E+09,9E+09]];
    CONST robtarget Target_9370:=[[68.835966618,63.302230963,30.312431948],[0.692516727,0.060687774,-0.040025666,0.717729422],[0,0,0,0],[9E+09,9E+09,9E+09,9E+09,9E+09,9E+09]];
    CONST robtarget Target_9380:=[[69.483445882,62.858623808,30.294039527],[0.692516726,0.060687774,-0.040025666,0.717729422],[0,0,0,0],[9E+09,9E+09,9E+09,9E+09,9E+09,9E+09]];
    CONST robtarget Target_9390:=[[70.17127725,62.480642126,30.274730357],[0.692516726,0.060687774,-0.040025666,0.717729422],[0,0,0,0],[9E+09,9E+09,9E+09,9E+09,9E+09,9E+09]];
    CONST robtarget Target_9400:=[[70.892836529,62.171926087,30.254690394],[0.692516726,0.060687774,-0.040025666,0.717729422],[0,0,0,0],[9E+09,9E+09,9E+09,9E+09,9E+09,9E+09]];
    CONST robtarget Target_9410:=[[71.64117471,61.935448798,30.234112635],[0.692516727,0.060687774,-0.040025666,0.717729422],[0,0,0,0],[9E+09,9E+09,9E+09,9E+09,9E+09,9E+09]];
    CONST robtarget Target_9420:=[[72.409084886,61.77348766,30.213195255],[0.692516726,0.060687774,-0.040025666,0.717729422],[0,0,0,0],[9E+09,9E+09,9E+09,9E+09,9E+09,9E+09]];
    CONST robtarget Target_9430:=[[73.189171664,61.68760245,30.1921397],[0.692516726,0.060687774,-0.040025667,0.717729423],[0,0,0,0],[9E+09,9E+09,9E+09,9E+09,9E+09,9E+09]];
    CONST robtarget Target_9440:=[[73.97392238,61.67862029,30.171148745],[0.692516726,0.060687774,-0.040025666,0.717729422],[0,0,0,0],[9E+09,9E+09,9E+09,9E+09,9E+09,9E+09]];
    CONST robtarget Target_9450:=[[127.916541834,63.711021485,28.734781164],[0.692516726,0.060687774,-0.040025667,0.717729422],[0,0,0,0],[9E+09,9E+09,9E+09,9E+09,9E+09,9E+09]];
    CONST robtarget Target_9460:=[[128.698398911,63.779028876,28.714056965],[0.692516726,0.060687774,-0.040025667,0.717729422],[0,0,0,0],[9E+09,9E+09,9E+09,9E+09,9E+09,9E+09]];
    CONST robtarget Target_9470:=[[129.469832636,63.923370871,28.693799107],[0.692516726,0.060687774,-0.040025666,0.717729422],[0,0,0,0],[9E+09,9E+09,9E+09,9E+09,9E+09,9E+09]];
    CONST robtarget Target_9480:=[[130.223413683,64.142657378,28.674202684],[0.692516726,0.060687774,-0.040025667,0.717729422],[0,0,0,0],[9E+09,9E+09,9E+09,9E+09,9E+09,9E+09]];
    CONST robtarget Target_9490:=[[130.951884654,64.434776547,28.65545642],[0.692516726,0.060687774,-0.040025666,0.717729422],[0,0,0,0],[9E+09,9E+09,9E+09,9E+09,9E+09,9E+09]];
    CONST robtarget Target_9500:=[[131.648229974,64.796915112,28.637740852],[0.692516726,0.060687774,-0.040025667,0.717729422],[0,0,0,0],[9E+09,9E+09,9E+09,9E+09,9E+09,9E+09]];
    CONST robtarget Target_9510:=[[132.305743457,65.225585479,28.621226591],[0.692516726,0.060687774,-0.040025666,0.717729422],[0,0,0,0],[9E+09,9E+09,9E+09,9E+09,9E+09,9E+09]];
    CONST robtarget Target_9520:=[[132.918092891,65.71665932,28.606072679],[0.692516726,0.060687774,-0.040025667,0.717729422],[0,0,0,0],[9E+09,9E+09,9E+09,9E+09,9E+09,9E+09]];
    CONST robtarget Target_9530:=[[133.479381014,66.265407323,28.592425054],[0.692516726,0.060687774,-0.040025666,0.717729422],[0,0,0,0],[9E+09,9E+09,9E+09,9E+09,9E+09,9E+09]];
    CONST robtarget Target_9540:=[[133.984202314,66.866544747,28.580415153],[0.692516726,0.060687774,-0.040025667,0.717729422],[0,0,0,0],[9E+09,9E+09,9E+09,9E+09,9E+09,9E+09]];
    CONST robtarget Target_9550:=[[134.427695089,67.514282309,28.570158635],[0.692516726,0.060687774,-0.040025667,0.717729422],[0,0,0,0],[9E+09,9E+09,9E+09,9E+09,9E+09,9E+09]];
    CONST robtarget Target_9560:=[[134.805588258,68.202381942,28.561754279],[0.692516726,0.060687774,-0.040025666,0.717729422],[0,0,0,0],[9E+09,9E+09,9E+09,9E+09,9E+09,9E+09]];
    CONST robtarget Target_9570:=[[135.114242504,68.924216872,28.555283021],[0.692516726,0.060687774,-0.040025667,0.717729422],[0,0,0,0],[9E+09,9E+09,9E+09,9E+09,9E+09,9E+09]];
    CONST robtarget Target_9580:=[[135.350685319,69.672835431,28.550807184],[0.692516726,0.060687774,-0.040025667,0.717729422],[0,0,0,0],[9E+09,9E+09,9E+09,9E+09,9E+09,9E+09]];
    CONST robtarget Target_9590:=[[135.512639628,70.441028015,28.548369872],[0.692516726,0.060687774,-0.040025667,0.717729422],[0,0,0,0],[9E+09,9E+09,9E+09,9E+09,9E+09,9E+09]];
    CONST robtarget Target_9600:=[[135.598545725,71.221396511,28.547994559],[0.692516726,0.060687774,-0.040025667,0.717729422],[0,0,0,0],[9E+09,9E+09,9E+09,9E+09,9E+09,9E+09]];
    CONST robtarget Target_9610:=[[135.607576284,72.006425541,28.549684858],[0.692516726,0.060687774,-0.040025667,0.717729422],[0,0,0,0],[9E+09,9E+09,9E+09,9E+09,9E+09,9E+09]];
    CONST robtarget Target_9620:=[[134.827212856,92.769146359,28.621624089],[0.692516726,0.060687774,-0.040025667,0.717729422],[0,0,0,0],[9E+09,9E+09,9E+09,9E+09,9E+09,9E+09]];
    CONST robtarget Target_9630:=[[135.609069933,92.837153751,28.60089989],[0.692516726,0.060687774,-0.040025667,0.717729422],[0,0,0,0],[9E+09,9E+09,9E+09,9E+09,9E+09,9E+09]];
    CONST robtarget Target_9640:=[[136.380503658,92.981495746,28.580642032],[0.692516726,0.060687774,-0.040025666,0.717729422],[0,0,0,0],[9E+09,9E+09,9E+09,9E+09,9E+09,9E+09]];
    CONST robtarget Target_9650:=[[137.134084705,93.200782252,28.561045609],[0.692516726,0.060687774,-0.040025667,0.717729422],[0,0,0,0],[9E+09,9E+09,9E+09,9E+09,9E+09,9E+09]];
    CONST robtarget Target_9660:=[[137.862555676,93.492901421,28.542299345],[0.692516726,0.060687774,-0.040025666,0.717729422],[0,0,0,0],[9E+09,9E+09,9E+09,9E+09,9E+09,9E+09]];
    CONST robtarget Target_9670:=[[138.558900996,93.855039986,28.524583777],[0.692516726,0.060687774,-0.040025667,0.717729422],[0,0,0,0],[9E+09,9E+09,9E+09,9E+09,9E+09,9E+09]];
    CONST robtarget Target_9680:=[[139.216414479,94.283710353,28.508069516],[0.692516726,0.060687774,-0.040025666,0.717729422],[0,0,0,0],[9E+09,9E+09,9E+09,9E+09,9E+09,9E+09]];
    CONST robtarget Target_9690:=[[139.828763913,94.774784193,28.492915604],[0.692516726,0.060687774,-0.040025667,0.717729422],[0,0,0,0],[9E+09,9E+09,9E+09,9E+09,9E+09,9E+09]];
    CONST robtarget Target_9700:=[[140.390052036,95.323532198,28.479267979],[0.692516726,0.060687774,-0.040025666,0.717729422],[0,0,0,0],[9E+09,9E+09,9E+09,9E+09,9E+09,9E+09]];
    CONST robtarget Target_9710:=[[140.894873336,95.924669621,28.467258078],[0.692516726,0.060687774,-0.040025667,0.717729422],[0,0,0,0],[9E+09,9E+09,9E+09,9E+09,9E+09,9E+09]];
    CONST robtarget Target_9720:=[[141.338366111,96.572407183,28.45700156],[0.692516726,0.060687774,-0.040025667,0.717729422],[0,0,0,0],[9E+09,9E+09,9E+09,9E+09,9E+09,9E+09]];
    CONST robtarget Target_9730:=[[141.71625928,97.260506816,28.448597204],[0.692516726,0.060687774,-0.040025666,0.717729422],[0,0,0,0],[9E+09,9E+09,9E+09,9E+09,9E+09,9E+09]];
    CONST robtarget Target_9740:=[[142.024913526,97.982341745,28.442125946],[0.692516726,0.060687774,-0.040025667,0.717729422],[0,0,0,0],[9E+09,9E+09,9E+09,9E+09,9E+09,9E+09]];
    CONST robtarget Target_9750:=[[142.261356341,98.730960305,28.437650109],[0.692516726,0.060687774,-0.040025667,0.717729422],[0,0,0,0],[9E+09,9E+09,9E+09,9E+09,9E+09,9E+09]];
    CONST robtarget Target_9760:=[[142.42331065,99.49915289,28.435212797],[0.692516726,0.060687774,-0.040025667,0.717729422],[0,0,0,0],[9E+09,9E+09,9E+09,9E+09,9E+09,9E+09]];
    CONST robtarget Target_9770:=[[142.509216747,100.279521384,28.434837484],[0.692516726,0.060687774,-0.040025667,0.717729422],[0,0,0,0],[9E+09,9E+09,9E+09,9E+09,9E+09,9E+09]];
    CONST robtarget Target_9780:=[[142.518247306,101.064550415,28.436527783],[0.692516726,0.060687774,-0.040025667,0.717729422],[0,0,0,0],[9E+09,9E+09,9E+09,9E+09,9E+09,9E+09]];
    CONST robtarget Target_9790:=[[142.45031536,101.846679721,28.440267416],[0.692516726,0.060687774,-0.040025667,0.717729422],[0,0,0,0],[9E+09,9E+09,9E+09,9E+09,9E+09,9E+09]];
    CONST robtarget Target_9800:=[[142.306075129,102.618376971,28.446020368],[0.692516726,0.060687774,-0.040025667,0.717729422],[0,0,0,0],[9E+09,9E+09,9E+09,9E+09,9E+09,9E+09]];
    CONST robtarget Target_9810:=[[142.086915728,103.372210298,28.453731236],[0.692516726,0.060687774,-0.040025666,0.717729422],[0,0,0,0],[9E+09,9E+09,9E+09,9E+09,9E+09,9E+09]];
    CONST robtarget Target_9820:=[[141.794947779,104.100919875,28.463325759],[0.692516726,0.060687774,-0.040025666,0.717729422],[0,0,0,0],[9E+09,9E+09,9E+09,9E+09,9E+09,9E+09]];
    CONST robtarget Target_9830:=[[141.432983095,104.797487831,28.474711537],[0.692516726,0.060687774,-0.040025667,0.717729422],[0,0,0,0],[9E+09,9E+09,9E+09,9E+09,9E+09,9E+09]];
    CONST robtarget Target_9840:=[[141.004507592,105.455205835,28.487778919],[0.692516726,0.060687774,-0.040025667,0.717729422],[0,0,0,0],[9E+09,9E+09,9E+09,9E+09,9E+09,9E+09]];
    CONST robtarget Target_9850:=[[140.513647725,106.067739704,28.502402059],[0.692516726,0.060687774,-0.040025667,0.717729422],[0,0,0,0],[9E+09,9E+09,9E+09,9E+09,9E+09,9E+09]];
    CONST robtarget Target_9860:=[[139.965130742,106.629190402,28.518440127],[0.692516726,0.060687774,-0.040025667,0.717729422],[0,0,0,0],[9E+09,9E+09,9E+09,9E+09,9E+09,9E+09]];
    CONST robtarget Target_9870:=[[139.364239161,107.13415085,28.535738668],[0.692516726,0.060687774,-0.040025666,0.717729422],[0,0,0,0],[9E+09,9E+09,9E+09,9E+09,9E+09,9E+09]];
    CONST robtarget Target_9880:=[[138.716759897,107.577758005,28.554131089],[0.692516726,0.060687774,-0.040025667,0.717729422],[0,0,0,0],[9E+09,9E+09,9E+09,9E+09,9E+09,9E+09]];
    CONST robtarget Target_9890:=[[138.02892853,107.955739687,28.573440259],[0.692516726,0.060687774,-0.040025667,0.717729422],[0,0,0,0],[9E+09,9E+09,9E+09,9E+09,9E+09,9E+09]];
    CONST robtarget Target_9900:=[[137.30736925,108.264455725,28.593480222],[0.692516726,0.060687774,-0.040025667,0.717729422],[0,0,0,0],[9E+09,9E+09,9E+09,9E+09,9E+09,9E+09]];
    CONST robtarget Target_9910:=[[136.559031069,108.500933016,28.614057981],[0.692516726,0.060687774,-0.040025666,0.717729422],[0,0,0,0],[9E+09,9E+09,9E+09,9E+09,9E+09,9E+09]];
    CONST robtarget Target_9920:=[[135.791120893,108.662894152,28.634975361],[0.692516726,0.060687774,-0.040025667,0.717729422],[0,0,0,0],[9E+09,9E+09,9E+09,9E+09,9E+09,9E+09]];
    CONST robtarget Target_9930:=[[135.011034116,108.748779362,28.656030917],[0.692516726,0.060687774,-0.040025666,0.717729422],[0,0,0,0],[9E+09,9E+09,9E+09,9E+09,9E+09,9E+09]];
    CONST robtarget Target_9940:=[[134.226283399,108.757761523,28.677021871],[0.692516726,0.060687774,-0.040025667,0.717729422],[0,0,0,0],[9E+09,9E+09,9E+09,9E+09,9E+09,9E+09]];
    CONST robtarget Target_9950:=[[133.579439368,125.968001721,28.736652372],[0.692516726,0.060687774,-0.040025667,0.717729422],[0,0,0,0],[9E+09,9E+09,9E+09,9E+09,9E+09,9E+09]];
    CONST robtarget Target_9960:=[[133.511507422,126.750131026,28.740392005],[0.692516726,0.060687774,-0.040025667,0.717729422],[0,0,0,0],[9E+09,9E+09,9E+09,9E+09,9E+09,9E+09]];
    CONST robtarget Target_9970:=[[133.367267191,127.521828277,28.746144958],[0.692516726,0.060687774,-0.040025667,0.717729422],[0,0,0,0],[9E+09,9E+09,9E+09,9E+09,9E+09,9E+09]];
    CONST robtarget Target_9980:=[[133.14810779,128.275661604,28.753855826],[0.692516726,0.060687774,-0.040025666,0.717729422],[0,0,0,0],[9E+09,9E+09,9E+09,9E+09,9E+09,9E+09]];
    CONST robtarget Target_9990:=[[132.856139841,129.00437118,28.763450349],[0.692516726,0.060687774,-0.040025666,0.717729422],[0,0,0,0],[9E+09,9E+09,9E+09,9E+09,9E+09,9E+09]];
    CONST robtarget Target_10000:=[[132.494175157,129.700939137,28.774836127],[0.692516726,0.060687774,-0.040025667,0.717729422],[0,0,0,0],[9E+09,9E+09,9E+09,9E+09,9E+09,9E+09]];
    CONST robtarget Target_10010:=[[132.065699654,130.358657141,28.787903509],[0.692516726,0.060687774,-0.040025667,0.717729422],[0,0,0,0],[9E+09,9E+09,9E+09,9E+09,9E+09,9E+09]];
    CONST robtarget Target_10020:=[[131.574839787,130.97119101,28.802526648],[0.692516726,0.060687774,-0.040025667,0.717729422],[0,0,0,0],[9E+09,9E+09,9E+09,9E+09,9E+09,9E+09]];
    CONST robtarget Target_10030:=[[131.026322804,131.532641707,28.818564716],[0.692516726,0.060687774,-0.040025667,0.717729422],[0,0,0,0],[9E+09,9E+09,9E+09,9E+09,9E+09,9E+09]];
    CONST robtarget Target_10040:=[[130.425431223,132.037602155,28.835863258],[0.692516726,0.060687774,-0.040025666,0.717729422],[0,0,0,0],[9E+09,9E+09,9E+09,9E+09,9E+09,9E+09]];
    CONST robtarget Target_10050:=[[129.777951959,132.481209311,28.854255678],[0.692516726,0.060687774,-0.040025667,0.717729422],[0,0,0,0],[9E+09,9E+09,9E+09,9E+09,9E+09,9E+09]];
    CONST robtarget Target_10060:=[[129.090120592,132.859190992,28.873564849],[0.692516726,0.060687774,-0.040025667,0.717729422],[0,0,0,0],[9E+09,9E+09,9E+09,9E+09,9E+09,9E+09]];
    CONST robtarget Target_10070:=[[128.368561312,133.167907031,28.893604812],[0.692516726,0.060687774,-0.040025667,0.717729422],[0,0,0,0],[9E+09,9E+09,9E+09,9E+09,9E+09,9E+09]];
    CONST robtarget Target_10080:=[[127.620223131,133.404384321,28.91418257],[0.692516726,0.060687774,-0.040025666,0.717729422],[0,0,0,0],[9E+09,9E+09,9E+09,9E+09,9E+09,9E+09]];
    CONST robtarget Target_10090:=[[126.852312954,133.566345459,28.935099951],[0.692516726,0.060687774,-0.040025667,0.717729422],[0,0,0,0],[9E+09,9E+09,9E+09,9E+09,9E+09,9E+09]];
    CONST robtarget Target_10100:=[[126.072226178,133.652230668,28.956155506],[0.692516726,0.060687774,-0.040025666,0.717729422],[0,0,0,0],[9E+09,9E+09,9E+09,9E+09,9E+09,9E+09]];
    CONST robtarget Target_10110:=[[125.287475461,133.661212829,28.977146461],[0.692516726,0.060687774,-0.040025667,0.717729422],[0,0,0,0],[9E+09,9E+09,9E+09,9E+09,9E+09,9E+09]];
    CONST robtarget Target_10120:=[[103.310852721,132.833197528,29.562333253],[0.692516726,0.060687774,-0.040025667,0.717729422],[0,0,0,0],[9E+09,9E+09,9E+09,9E+09,9E+09,9E+09]];
    CONST robtarget Target_10130:=[[102.509529144,132.906987315,-0.426872065],[0.692516726,0.060687774,-0.040025667,0.717729422],[0,0,0,0],[9E+09,9E+09,9E+09,9E+09,9E+09,9E+09]];
    CONST robtarget Target_10140:=[[110.727588271,100.564281,-0.726042579],[0.692516726,0.060687774,-0.040025667,0.717729422],[0,0,0,0],[9E+09,9E+09,9E+09,9E+09,9E+09,9E+09]];
    CONST robtarget Target_10150:=[[111.528911848,100.490491212,29.263162739],[0.692516726,0.060687774,-0.040025667,0.717729422],[0,0,0,0],[9E+09,9E+09,9E+09,9E+09,9E+09,9E+09]];
    CONST robtarget Target_10160:=[[110.685548697,100.498289722,29.285716929],[0.692516726,0.060687774,-0.040025667,0.717729422],[0,0,0,0],[9E+09,9E+09,9E+09,9E+09,9E+09,9E+09]];
    CONST robtarget Target_10170:=[[109.846626496,100.585055744,29.308346758],[0.692516726,0.060687774,-0.040025667,0.717729422],[0,0,0,0],[9E+09,9E+09,9E+09,9E+09,9E+09,9E+09]];
    CONST robtarget Target_10180:=[[109.019517721,100.750026775,29.330853354],[0.692516726,0.060687774,-0.040025667,0.717729422],[0,0,0,0],[9E+09,9E+09,9E+09,9E+09,9E+09,9E+09]];
    CONST robtarget Target_10190:=[[108.211491036,100.991753042,29.353038929],[0.692516726,0.060687774,-0.040025667,0.717729422],[0,0,0,0],[9E+09,9E+09,9E+09,9E+09,9E+09,9E+09]];
    CONST robtarget Target_10200:=[[107.429647407,101.308110249,29.374708515],[0.692516726,0.060687774,-0.040025666,0.717729422],[0,0,0,0],[9E+09,9E+09,9E+09,9E+09,9E+09,9E+09]];
    CONST robtarget Target_10210:=[[106.680857706,101.696318234,29.395671679],[0.692516726,0.060687774,-0.040025666,0.717729422],[0,0,0,0],[9E+09,9E+09,9E+09,9E+09,9E+09,9E+09]];
    CONST robtarget Target_10220:=[[105.971702321,102.152965415,29.415744196],[0.692516726,0.060687774,-0.040025666,0.717729422],[0,0,0,0],[9E+09,9E+09,9E+09,9E+09,9E+09,9E+09]];
    CONST robtarget Target_10230:=[[105.308413336,102.674038757,29.434749667],[0.692516726,0.060687774,-0.040025667,0.717729422],[0,0,0,0],[9E+09,9E+09,9E+09,9E+09,9E+09,9E+09]];
    CONST robtarget Target_10240:=[[104.696819761,103.254959051,29.452521073],[0.692516726,0.060687774,-0.040025667,0.717729422],[0,0,0,0],[9E+09,9E+09,9E+09,9E+09,9E+09,9E+09]];
    CONST robtarget Target_10250:=[[104.142296299,103.890621146,29.468902237],[0.692516726,0.060687774,-0.040025667,0.717729422],[0,0,0,0],[9E+09,9E+09,9E+09,9E+09,9E+09,9E+09]];
    CONST robtarget Target_10260:=[[103.649716123,104.575438823,29.483749202],[0.692516726,0.060687774,-0.040025666,0.717729422],[0,0,0,0],[9E+09,9E+09,9E+09,9E+09,9E+09,9E+09]];
    CONST robtarget Target_10270:=[[103.223408046,105.303393879,29.49693149],[0.692516726,0.060687774,-0.040025666,0.717729422],[0,0,0,0],[9E+09,9E+09,9E+09,9E+09,9E+09,9E+09]];
    CONST robtarget Target_10280:=[[102.867118479,106.068089018,29.508333257],[0.692516726,0.060687774,-0.040025667,0.717729422],[0,0,0,0],[9E+09,9E+09,9E+09,9E+09,9E+09,9E+09]];
    CONST robtarget Target_10290:=[[102.583978506,106.862804074,29.517854303],[0.692516726,0.060687774,-0.040025666,0.717729422],[0,0,0,0],[9E+09,9E+09,9E+09,9E+09,9E+09,9E+09]];
    CONST robtarget Target_10300:=[[102.376476372,107.680555058,29.525410956],[0.692516726,0.060687774,-0.040025667,0.717729422],[0,0,0,0],[9E+09,9E+09,9E+09,9E+09,9E+09,9E+09]];
    CONST robtarget Target_10310:=[[102.246435614,108.514155549,29.530936808],[0.692516726,0.060687774,-0.040025666,0.717729422],[0,0,0,0],[9E+09,9E+09,9E+09,9E+09,9E+09,9E+09]];
    CONST robtarget Target_10320:=[[102.194999034,109.356279835,29.534383299],[0.692516726,0.060687774,-0.040025666,0.717729422],[0,0,0,0],[9E+09,9E+09,9E+09,9E+09,9E+09,9E+09]];
    CONST robtarget Target_10330:=[[102.222618659,110.199527297,29.53572014],[0.692516726,0.060687774,-0.040025667,0.717729422],[0,0,0,0],[9E+09,9E+09,9E+09,9E+09,9E+09,9E+09]];
    CONST robtarget Target_10340:=[[102.329051766,111.036487446,29.534935583],[0.692516726,0.060687774,-0.040025667,0.717729422],[0,0,0,0],[9E+09,9E+09,9E+09,9E+09,9E+09,9E+09]];
    CONST robtarget Target_10350:=[[102.513363018,111.859805046,29.532036522],[0.692516726,0.060687774,-0.040025666,0.717729422],[0,0,0,0],[9E+09,9E+09,9E+09,9E+09,9E+09,9E+09]];
    CONST robtarget Target_10360:=[[102.77393268,112.662244752,29.527048435],[0.692516726,0.060687774,-0.040025666,0.717729422],[0,0,0,0],[9E+09,9E+09,9E+09,9E+09,9E+09,9E+09]];
    CONST robtarget Target_10370:=[[103.108470858,113.436754696,29.520015158],[0.692516726,0.060687774,-0.040025667,0.717729422],[0,0,0,0],[9E+09,9E+09,9E+09,9E+09,9E+09,9E+09]];
    CONST robtarget Target_10380:=[[103.514037617,114.176528456,29.510998498],[0.692516726,0.060687774,-0.040025667,0.717729422],[0,0,0,0],[9E+09,9E+09,9E+09,9E+09,9E+09,9E+09]];
    CONST robtarget Target_10390:=[[103.987068821,114.875064874,29.500077695],[0.692516726,0.060687774,-0.040025666,0.717729422],[0,0,0,0],[9E+09,9E+09,9E+09,9E+09,9E+09,9E+09]];
    CONST robtarget Target_10400:=[[104.523407458,115.526225188,29.487348721],[0.692516726,0.060687774,-0.040025667,0.717729422],[0,0,0,0],[9E+09,9E+09,9E+09,9E+09,9E+09,9E+09]];
    CONST robtarget Target_10410:=[[105.118340161,116.124286975,29.472923439],[0.692516726,0.060687774,-0.040025667,0.717729422],[0,0,0,0],[9E+09,9E+09,9E+09,9E+09,9E+09,9E+09]];
    CONST robtarget Target_10420:=[[105.766638643,116.663994448,29.456928619],[0.692516726,0.060687774,-0.040025666,0.717729422],[0,0,0,0],[9E+09,9E+09,9E+09,9E+09,9E+09,9E+09]];
    CONST robtarget Target_10430:=[[106.462605632,117.140604638,29.439504823],[0.692516726,0.060687774,-0.040025666,0.717729422],[0,0,0,0],[9E+09,9E+09,9E+09,9E+09,9E+09,9E+09]];
    CONST robtarget Target_10440:=[[107.200124946,117.54992908,29.420805172],[0.692516726,0.060687774,-0.040025666,0.717729422],[0,0,0,0],[9E+09,9E+09,9E+09,9E+09,9E+09,9E+09]];
    CONST robtarget Target_10450:=[[107.972715238,117.888370611,29.400994001],[0.692516726,0.060687774,-0.040025667,0.717729422],[0,0,0,0],[9E+09,9E+09,9E+09,9E+09,9E+09,9E+09]];
    CONST robtarget Target_10460:=[[108.773586957,118.152955,29.38024541],[0.692516726,0.060687774,-0.040025667,0.717729422],[0,0,0,0],[9E+09,9E+09,9E+09,9E+09,9E+09,9E+09]];
    CONST robtarget Target_10470:=[[109.595702013,118.341357067,29.358741738],[0.692516726,0.060687774,-0.040025667,0.717729422],[0,0,0,0],[9E+09,9E+09,9E+09,9E+09,9E+09,9E+09]];
    CONST robtarget Target_10480:=[[110.43183563,118.451921127,29.336671961],[0.692516726,0.060687774,-0.040025666,0.717729422],[0,0,0,0],[9E+09,9E+09,9E+09,9E+09,9E+09,9E+09]];
    CONST robtarget Target_10490:=[[111.274639836,118.483675541,29.314230028],[0.692516726,0.060687774,-0.040025666,0.717729422],[0,0,0,0],[9E+09,9E+09,9E+09,9E+09,9E+09,9E+09]];
    CONST robtarget Target_10500:=[[112.116708037,118.43634125,29.29161316],[0.692516726,0.060687774,-0.040025667,0.717729422],[0,0,0,0],[9E+09,9E+09,9E+09,9E+09,9E+09,9E+09]];
    CONST robtarget Target_10510:=[[112.950640107,118.310334228,29.269020115],[0.692516726,0.060687774,-0.040025666,0.717729422],[0,0,0,0],[9E+09,9E+09,9E+09,9E+09,9E+09,9E+09]];
    CONST robtarget Target_10520:=[[113.769107421,118.10676183,29.246649442],[0.692516726,0.060687774,-0.040025667,0.717729422],[0,0,0,0],[9E+09,9E+09,9E+09,9E+09,9E+09,9E+09]];
    CONST robtarget Target_10530:=[[114.564917259,117.827413059,29.224697734],[0.692516726,0.060687774,-0.040025666,0.717729422],[0,0,0,0],[9E+09,9E+09,9E+09,9E+09,9E+09,9E+09]];
    CONST robtarget Target_10540:=[[115.331076017,117.474742839,29.203357904],[0.692516726,0.060687774,-0.040025667,0.717729422],[0,0,0,0],[9E+09,9E+09,9E+09,9E+09,9E+09,9E+09]];
    CONST robtarget Target_10550:=[[116.060850661,117.051850452,29.182817488],[0.692516726,0.060687774,-0.040025667,0.717729422],[0,0,0,0],[9E+09,9E+09,9E+09,9E+09,9E+09,9E+09]];
    CONST robtarget Target_10560:=[[116.747827907,116.562452289,29.163256994],[0.692516726,0.060687774,-0.040025666,0.717729422],[0,0,0,0],[9E+09,9E+09,9E+09,9E+09,9E+09,9E+09]];
    CONST robtarget Target_10570:=[[117.385970576,116.0108492,29.144848322],[0.692516726,0.060687774,-0.040025667,0.717729422],[0,0,0,0],[9E+09,9E+09,9E+09,9E+09,9E+09,9E+09]];
    CONST robtarget Target_10580:=[[117.969670644,115.401888691,29.127753248],[0.692516726,0.060687774,-0.040025666,0.717729422],[0,0,0,0],[9E+09,9E+09,9E+09,9E+09,9E+09,9E+09]];
    CONST robtarget Target_10590:=[[118.493798537,114.740922331,29.112122004],[0.692516726,0.060687774,-0.040025667,0.717729422],[0,0,0,0],[9E+09,9E+09,9E+09,9E+09,9E+09,9E+09]];
    CONST robtarget Target_10600:=[[118.953748198,114.033758715,29.098091957],[0.692516726,0.060687774,-0.040025666,0.717729422],[0,0,0,0],[9E+09,9E+09,9E+09,9E+09,9E+09,9E+09]];
    CONST robtarget Target_10610:=[[119.345477572,113.286612423,29.085786404],[0.692516726,0.060687774,-0.040025666,0.717729422],[0,0,0,0],[9E+09,9E+09,9E+09,9E+09,9E+09,9E+09]];
    CONST robtarget Target_10620:=[[119.665544131,112.506049402,29.075313487],[0.692516726,0.060687774,-0.040025666,0.717729422],[0,0,0,0],[9E+09,9E+09,9E+09,9E+09,9E+09,9E+09]];
    CONST robtarget Target_10630:=[[119.911135115,111.69892927,29.066765242],[0.692516726,0.060687774,-0.040025666,0.717729422],[0,0,0,0],[9E+09,9E+09,9E+09,9E+09,9E+09,9E+09]];
    CONST robtarget Target_10640:=[[120.080092264,110.872345026,29.060216791],[0.692516726,0.060687774,-0.040025667,0.717729422],[0,0,0,0],[9E+09,9E+09,9E+09,9E+09,9E+09,9E+09]];
    CONST robtarget Target_10650:=[[120.170930774,110.033560722,29.055725684],[0.692516726,0.060687774,-0.040025667,0.717729422],[0,0,0,0],[9E+09,9E+09,9E+09,9E+09,9E+09,9E+09]];
    CONST robtarget Target_10660:=[[120.182852355,109.189947626,29.053331386],[0.692516726,0.060687774,-0.040025667,0.717729422],[0,0,0,0],[9E+09,9E+09,9E+09,9E+09,9E+09,9E+09]];
    CONST robtarget Target_10670:=[[120.115752238,108.34891944,29.053054941],[0.692516726,0.060687774,-0.040025667,0.717729422],[0,0,0,0],[9E+09,9E+09,9E+09,9E+09,9E+09,9E+09]];
    CONST robtarget Target_10680:=[[119.970220103,107.517867149,29.054898776],[0.692516726,0.060687774,-0.040025667,0.717729422],[0,0,0,0],[9E+09,9E+09,9E+09,9E+09,9E+09,9E+09]];
    CONST robtarget Target_10690:=[[119.747534891,106.704094071,29.058846689],[0.692516726,0.060687774,-0.040025667,0.717729422],[0,0,0,0],[9E+09,9E+09,9E+09,9E+09,9E+09,9E+09]];
    CONST robtarget Target_10700:=[[119.449653567,105.914751672,29.064863985],[0.692516726,0.060687774,-0.040025667,0.717729422],[0,0,0,0],[9E+09,9E+09,9E+09,9E+09,9E+09,9E+09]];
    CONST robtarget Target_10710:=[[119.079193923,105.156776724,29.072897783],[0.692516726,0.060687774,-0.040025666,0.717729422],[0,0,0,0],[9E+09,9E+09,9E+09,9E+09,9E+09,9E+09]];
    CONST robtarget Target_10720:=[[118.639411573,104.436830335,29.082877483],[0.692516726,0.060687774,-0.040025667,0.717729422],[0,0,0,0],[9E+09,9E+09,9E+09,9E+09,9E+09,9E+09]];
    CONST robtarget Target_10730:=[[118.134171339,103.761239422,29.094715383],[0.692516726,0.060687774,-0.040025667,0.717729422],[0,0,0,0],[9E+09,9E+09,9E+09,9E+09,9E+09,9E+09]];
    CONST robtarget Target_10740:=[[117.567913289,103.135941101,29.10830745],[0.692516726,0.060687774,-0.040025667,0.717729422],[0,0,0,0],[9E+09,9E+09,9E+09,9E+09,9E+09,9E+09]];
    CONST robtarget Target_10750:=[[116.945613722,102.566430517,29.123534237],[0.692516726,0.060687774,-0.040025666,0.717729422],[0,0,0,0],[9E+09,9E+09,9E+09,9E+09,9E+09,9E+09]];
    CONST robtarget Target_10760:=[[116.272741427,102.057712548,29.140261931],[0.692516726,0.060687774,-0.040025667,0.717729422],[0,0,0,0],[9E+09,9E+09,9E+09,9E+09,9E+09,9E+09]];
    CONST robtarget Target_10770:=[[115.55520963,101.614257828,29.158343528],[0.692516726,0.060687774,-0.040025667,0.717729422],[0,0,0,0],[9E+09,9E+09,9E+09,9E+09,9E+09,9E+09]];
    CONST robtarget Target_10780:=[[114.799324027,101.239963452,29.177620126],[0.692516726,0.060687774,-0.040025667,0.717729422],[0,0,0,0],[9E+09,9E+09,9E+09,9E+09,9E+09,9E+09]];
    CONST robtarget Target_10790:=[[114.011727368,100.938118732,29.197922322],[0.692516726,0.060687774,-0.040025667,0.717729422],[0,0,0,0],[9E+09,9E+09,9E+09,9E+09,9E+09,9E+09]];
    CONST robtarget Target_10800:=[[113.19934108,100.71137629,29.219071699],[0.692516726,0.060687774,-0.040025666,0.717729422],[0,0,0,0],[9E+09,9E+09,9E+09,9E+09,9E+09,9E+09]];
    CONST robtarget Target_10810:=[[112.369304442,100.561728748,29.240882395],[0.692516726,0.060687774,-0.040025666,0.717729422],[0,0,0,0],[9E+09,9E+09,9E+09,9E+09,9E+09,9E+09]];
    CONST robtarget Target_10820:=[[111.528911848,100.490491212,29.263162739],[0.692516726,0.060687774,-0.040025667,0.717729422],[0,0,0,0],[9E+09,9E+09,9E+09,9E+09,9E+09,9E+09]];
    CONST robtarget Target_10830:=[[110.727588271,100.564281,-0.726042579],[0.692516726,0.060687774,-0.040025667,0.717729422],[0,0,0,0],[9E+09,9E+09,9E+09,9E+09,9E+09,9E+09]];
    CONST robtarget Target_10840:=[[86.753090736,99.66099158,-0.087656987],[0.692516726,0.060687774,-0.040025667,0.717729422],[0,0,0,0],[9E+09,9E+09,9E+09,9E+09,9E+09,9E+09]];
    CONST robtarget Target_10850:=[[87.554414313,99.587201792,29.901548331],[0.692516726,0.060687774,-0.040025667,0.717729422],[0,0,0,0],[9E+09,9E+09,9E+09,9E+09,9E+09,9E+09]];
    CONST robtarget Target_10860:=[[86.711051162,99.595000302,29.92410252],[0.692516726,0.060687774,-0.040025667,0.717729422],[0,0,0,0],[9E+09,9E+09,9E+09,9E+09,9E+09,9E+09]];
    CONST robtarget Target_10870:=[[85.872128961,99.681766324,29.946732349],[0.692516726,0.060687774,-0.040025667,0.717729422],[0,0,0,0],[9E+09,9E+09,9E+09,9E+09,9E+09,9E+09]];
    CONST robtarget Target_10880:=[[85.045020186,99.846737355,29.969238946],[0.692516726,0.060687774,-0.040025667,0.717729422],[0,0,0,0],[9E+09,9E+09,9E+09,9E+09,9E+09,9E+09]];
    CONST robtarget Target_10890:=[[84.236993501,100.088463622,29.991424521],[0.692516726,0.060687774,-0.040025667,0.717729422],[0,0,0,0],[9E+09,9E+09,9E+09,9E+09,9E+09,9E+09]];
    CONST robtarget Target_10900:=[[83.455149872,100.404820829,30.013094107],[0.692516726,0.060687774,-0.040025666,0.717729422],[0,0,0,0],[9E+09,9E+09,9E+09,9E+09,9E+09,9E+09]];
    CONST robtarget Target_10910:=[[82.706360171,100.793028814,30.034057271],[0.692516726,0.060687774,-0.040025666,0.717729422],[0,0,0,0],[9E+09,9E+09,9E+09,9E+09,9E+09,9E+09]];
    CONST robtarget Target_10920:=[[81.997204786,101.249675995,30.054129787],[0.692516726,0.060687774,-0.040025666,0.717729422],[0,0,0,0],[9E+09,9E+09,9E+09,9E+09,9E+09,9E+09]];
    CONST robtarget Target_10930:=[[81.333915801,101.770749337,30.073135259],[0.692516726,0.060687774,-0.040025667,0.717729422],[0,0,0,0],[9E+09,9E+09,9E+09,9E+09,9E+09,9E+09]];
    CONST robtarget Target_10940:=[[80.722322226,102.351669631,30.090906665],[0.692516726,0.060687774,-0.040025667,0.717729422],[0,0,0,0],[9E+09,9E+09,9E+09,9E+09,9E+09,9E+09]];
    CONST robtarget Target_10950:=[[80.167798764,102.987331726,30.107287829],[0.692516726,0.060687774,-0.040025667,0.717729422],[0,0,0,0],[9E+09,9E+09,9E+09,9E+09,9E+09,9E+09]];
    CONST robtarget Target_10960:=[[79.675218588,103.672149403,30.122134793],[0.692516726,0.060687774,-0.040025666,0.717729422],[0,0,0,0],[9E+09,9E+09,9E+09,9E+09,9E+09,9E+09]];
    CONST robtarget Target_10970:=[[79.248910511,104.400104459,30.135317082],[0.692516726,0.060687774,-0.040025666,0.717729422],[0,0,0,0],[9E+09,9E+09,9E+09,9E+09,9E+09,9E+09]];
    CONST robtarget Target_10980:=[[78.892620944,105.164799598,30.146718849],[0.692516726,0.060687774,-0.040025667,0.717729422],[0,0,0,0],[9E+09,9E+09,9E+09,9E+09,9E+09,9E+09]];
    CONST robtarget Target_10990:=[[78.609480971,105.959514653,30.156239894],[0.692516726,0.060687774,-0.040025666,0.717729422],[0,0,0,0],[9E+09,9E+09,9E+09,9E+09,9E+09,9E+09]];
    CONST robtarget Target_11000:=[[78.401978837,106.777265638,30.163796547],[0.692516726,0.060687774,-0.040025667,0.717729422],[0,0,0,0],[9E+09,9E+09,9E+09,9E+09,9E+09,9E+09]];
    CONST robtarget Target_11010:=[[78.271938079,107.610866129,30.1693224],[0.692516726,0.060687774,-0.040025666,0.717729422],[0,0,0,0],[9E+09,9E+09,9E+09,9E+09,9E+09,9E+09]];
    CONST robtarget Target_11020:=[[78.220501499,108.452990415,30.172768891],[0.692516726,0.060687774,-0.040025666,0.717729422],[0,0,0,0],[9E+09,9E+09,9E+09,9E+09,9E+09,9E+09]];
    CONST robtarget Target_11030:=[[78.248121124,109.296237877,30.174105732],[0.692516726,0.060687774,-0.040025667,0.717729422],[0,0,0,0],[9E+09,9E+09,9E+09,9E+09,9E+09,9E+09]];
    CONST robtarget Target_11040:=[[78.354554231,110.133198026,30.173321174],[0.692516726,0.060687774,-0.040025667,0.717729422],[0,0,0,0],[9E+09,9E+09,9E+09,9E+09,9E+09,9E+09]];
    CONST robtarget Target_11050:=[[78.538865483,110.956515626,30.170422114],[0.692516726,0.060687774,-0.040025666,0.717729422],[0,0,0,0],[9E+09,9E+09,9E+09,9E+09,9E+09,9E+09]];
    CONST robtarget Target_11060:=[[78.799435145,111.758955332,30.165434027],[0.692516726,0.060687774,-0.040025666,0.717729422],[0,0,0,0],[9E+09,9E+09,9E+09,9E+09,9E+09,9E+09]];
    CONST robtarget Target_11070:=[[79.133973323,112.533465275,30.15840075],[0.692516726,0.060687774,-0.040025667,0.717729422],[0,0,0,0],[9E+09,9E+09,9E+09,9E+09,9E+09,9E+09]];
    CONST robtarget Target_11080:=[[79.539540081,113.273239036,30.14938409],[0.692516726,0.060687774,-0.040025667,0.717729422],[0,0,0,0],[9E+09,9E+09,9E+09,9E+09,9E+09,9E+09]];
    CONST robtarget Target_11090:=[[80.012571286,113.971775454,30.138463287],[0.692516726,0.060687774,-0.040025666,0.717729422],[0,0,0,0],[9E+09,9E+09,9E+09,9E+09,9E+09,9E+09]];
    CONST robtarget Target_11100:=[[80.548909923,114.622935767,30.125734313],[0.692516726,0.060687774,-0.040025667,0.717729422],[0,0,0,0],[9E+09,9E+09,9E+09,9E+09,9E+09,9E+09]];
    CONST robtarget Target_11110:=[[81.143842626,115.220997555,30.111309031],[0.692516726,0.060687774,-0.040025667,0.717729422],[0,0,0,0],[9E+09,9E+09,9E+09,9E+09,9E+09,9E+09]];
    CONST robtarget Target_11120:=[[81.792141108,115.760705028,30.09531421],[0.692516726,0.060687774,-0.040025666,0.717729422],[0,0,0,0],[9E+09,9E+09,9E+09,9E+09,9E+09,9E+09]];
    CONST robtarget Target_11130:=[[82.488108097,116.237315218,30.077890414],[0.692516726,0.060687774,-0.040025666,0.717729422],[0,0,0,0],[9E+09,9E+09,9E+09,9E+09,9E+09,9E+09]];
    CONST robtarget Target_11140:=[[83.225627411,116.646639659,30.059190764],[0.692516726,0.060687774,-0.040025666,0.717729422],[0,0,0,0],[9E+09,9E+09,9E+09,9E+09,9E+09,9E+09]];
    CONST robtarget Target_11150:=[[83.998217703,116.985081191,30.039379593],[0.692516726,0.060687774,-0.040025667,0.717729422],[0,0,0,0],[9E+09,9E+09,9E+09,9E+09,9E+09,9E+09]];
    CONST robtarget Target_11160:=[[84.799089422,117.24966558,30.018631001],[0.692516726,0.060687774,-0.040025667,0.717729422],[0,0,0,0],[9E+09,9E+09,9E+09,9E+09,9E+09,9E+09]];
    CONST robtarget Target_11170:=[[85.621204478,117.438067646,29.99712733],[0.692516726,0.060687774,-0.040025667,0.717729422],[0,0,0,0],[9E+09,9E+09,9E+09,9E+09,9E+09,9E+09]];
    CONST robtarget Target_11180:=[[86.457338095,117.548631706,29.975057552],[0.692516726,0.060687774,-0.040025666,0.717729422],[0,0,0,0],[9E+09,9E+09,9E+09,9E+09,9E+09,9E+09]];
    CONST robtarget Target_11190:=[[87.300142301,117.580386121,29.95261562],[0.692516726,0.060687774,-0.040025666,0.717729422],[0,0,0,0],[9E+09,9E+09,9E+09,9E+09,9E+09,9E+09]];
    CONST robtarget Target_11200:=[[88.142210502,117.53305183,29.929998752],[0.692516726,0.060687774,-0.040025667,0.717729422],[0,0,0,0],[9E+09,9E+09,9E+09,9E+09,9E+09,9E+09]];
